(* Logix 5000 project; controller R1USB70001_CWRU_GRID_20120217 vendor 1 type 14 code 54 rev 19.11; software revision 19.01 *)

TASK MainTask (continuous, watchdog 500 ms) : MainProgram

MODULES
   Local : vendor 1 type 14 code 54 (ICP 2, rev 19.11)
      CNB_GRID : vendor 1 type 12 code 21 (ICP 0, rev 20.1)
         ACNR_GP_SC_N2 : vendor 1 type 12 code 111 (ControlNet 2, rev 1.83, Output RPI 16 ms)
            IE4C_GP_SC_S4 : 1734-IE4C (PointIO 4, rev 3.1, Input RPI 16 ms)
            IB8_GP_SC_S11 : 1734-IB8 (PointIO 11, rev 3.22)
            IE4C_GP_SC_S8 : 1734-IE4C (PointIO 8, rev 3.1, Input RPI 16 ms)
            IE4C_GP_SC_S5 : 1734-IE4C (PointIO 5, rev 3.1, Input RPI 16 ms)
            IE4C_GP_SC_S6 : 1734-IE4C (PointIO 6, rev 3.1, Input RPI 16 ms)
            IE4C_GP_SC_S9 : 1734-IE4C (PointIO 9, rev 3.1, Input RPI 16 ms)
            IE4C_GP_SC_S1 : 1734-IE4C (PointIO 1, rev 3.1, Input RPI 16 ms)
            IB8_GP_SC_S10 : 1734-IB8 (PointIO 10, rev 3.22)
            IE4C_GP_SC_S2 : 1734-IE4C (PointIO 2, rev 3.1, Input RPI 16 ms)
            IE4C_GP_SC_S7 : 1734-IE4C (PointIO 7, rev 3.1, Input RPI 16 ms)
            IE4C_GP_SC_S3 : 1734-IE4C (PointIO 3, rev 3.1, Input RPI 16 ms)
            OB8_GP_SC_S19 : 1734-OB8 (PointIO 19, rev 3.22)
            OB8_GP_SC_S13 : 1734-OB8 (PointIO 13, rev 3.22)
            OB8_GP_SC_S18 : 1734-OB8 (PointIO 18, rev 3.22)
            OB8_GP_SC_S23 : 1734-OB8 (PointIO 23, rev 3.22)
            OB8_GP_SC_S12 : 1734-OB8 (PointIO 12, rev 3.22)
            OB8_GP_SC_S20 : 1734-OB8 (PointIO 20, rev 3.22)
            OB8_GP_SC_S17 : 1734-OB8 (PointIO 17, rev 3.22)
            OB8_GP_SC_S15 : 1734-OB8 (PointIO 15, rev 3.22)
            OB8_GP_SC_S21 : 1734-OB8 (PointIO 21, rev 3.22)
            OB8_GP_SC_S22 : 1734-OB8 (PointIO 22, rev 3.22)
            OB8_GP_SC_S14 : 1734-OB8 (PointIO 14, rev 3.22)
            OB8_GP_SC_S16 : 1734-OB8 (PointIO 16, rev 3.22)
      EN2T_GRID : 1756-EN2T (ICP 1, Ethernet 10.88.0.102, rev 4.3)
END_MODULES

VAR_GLOBAL   (* controller tags *)
   AP_GP_CH_ACAM : ALIAS FOR ACNR_GP_SC_N2:1:I.Ch1Data;
   AP_GP_CH_CS : ALIAS FOR ACNR_GP_SC_N2:12:O.1;
   AP_GP_SR_ACAM : ALIAS FOR ACNR_GP_SC_N2:1:I.Ch0Data;
   AP_GP_SR_ACVT : ALIAS FOR ACNR_GP_SC_N2:9:I.Ch1Data;
   AP_GP_SR_CS : ALIAS FOR ACNR_GP_SC_N2:12:O.0;
   BT_GP_CH1_CS : ALIAS FOR ACNR_GP_SC_N2:12:O.3;
   BT_GP_CH2_CS : ALIAS FOR ACNR_GP_SC_N2:12:O.4;
   BT_GP_L1_ACAM1 : ALIAS FOR ACNR_GP_SC_N2:1:I.Ch2Data;
   BT_GP_L1_ACAM2 : ALIAS FOR ACNR_GP_SC_N2:1:I.Ch3Data;
   BT_GP_L1_DCAM : ALIAS FOR ACNR_GP_SC_N2:2:I.Ch2Data;
   BT_GP_L1_DCVS : ALIAS FOR ACNR_GP_SC_N2:10:I.2;
   BT_GP_L2_ACAM1 : ALIAS FOR ACNR_GP_SC_N2:2:I.Ch0Data;
   BT_GP_L2_DCAM : ALIAS FOR ACNR_GP_SC_N2:2:I.Ch3Data;
   BT_GP_ML_ACVT : ALIAS FOR ACNR_GP_SC_N2:9:I.Ch2Data;
   BT_GP_SR1_CS : ALIAS FOR ACNR_GP_SC_N2:12:O.6;
   BT_GP_SR2_CS : ALIAS FOR ACNR_GP_SC_N2:12:O.7;
   BT_GP_SR3_CS : ALIAS FOR ACNR_GP_SC_N2:13:O.0;
   CAP3_3_USER : BOOL;
   CAP_10_USER : BOOL;
   CAP_11_USER : BOOL;
   CAP_12_USER : BOOL;
   CAP_13_USER : BOOL;
   CAP_14_USER : BOOL;
   CAP_15_USER : BOOL;
   CAP_16_USER : BOOL;
   CAP_17_USER : BOOL;
   CAP_18_USER : BOOL;
   CAP_19_USER : BOOL;
   CAP_1_USER : BOOL;
   CAP_20_USER : BOOL;
   CAP_21_USER : BOOL;
   CAP_22_USER : BOOL;
   CAP_23_USER : BOOL;
   CAP_24_USER : BOOL;
   CAP_25_USER : BOOL;
   CAP_26_USER : BOOL;
   CAP_27_USER : BOOL;
   CAP_28_USER : BOOL;
   CAP_29_USER : BOOL;
   CAP_2_USER : BOOL;
   CAP_30_USER : BOOL;
   CAP_31_USER : BOOL;
   CAP_32_USER : BOOL;
   CAP_33_USER : BOOL;
   CAP_34_USER : BOOL;
   CAP_35_USER : BOOL;
   CAP_36_USER : BOOL;
   CAP_37_USER : BOOL;
   CAP_38_USER : BOOL;
   CAP_39_USER : BOOL;
   CAP_3_USER : BOOL;
   CAP_40_USER : BOOL;
   CAP_41_USER : BOOL;
   CAP_42_USER : BOOL;
   CAP_43_USER : BOOL;
   CAP_44_USER : BOOL;
   CAP_45_USER : BOOL;
   CAP_46_USER : BOOL;
   CAP_47_USER : BOOL;
   CAP_48_USER : BOOL;
   CAP_49_USER : BOOL;
   CAP_4_USER : BOOL;
   CAP_50_USER : BOOL;
   CAP_5_USER : BOOL;
   CAP_6_USER : BOOL;
   CAP_7_USER : BOOL;
   CAP_8_USER : BOOL;
   CAP_9_USER : BOOL;
   CAP_MAIN_USER : BOOL;
   CAP_MORE : DINT;
   CB_GP_C10_CS : ALIAS FOR ACNR_GP_SC_N2:18:O.2;
   CB_GP_C11_CS : ALIAS FOR ACNR_GP_SC_N2:18:O.3;
   CB_GP_C12_CS : ALIAS FOR ACNR_GP_SC_N2:18:O.4;
   CB_GP_C13_CS : ALIAS FOR ACNR_GP_SC_N2:18:O.5;
   CB_GP_C14_CS : ALIAS FOR ACNR_GP_SC_N2:18:O.6;
   CB_GP_C15_CS : ALIAS FOR ACNR_GP_SC_N2:18:O.7;
   CB_GP_C16_CS : ALIAS FOR ACNR_GP_SC_N2:19:O.0;
   CB_GP_C17_CS : ALIAS FOR ACNR_GP_SC_N2:19:O.1;
   CB_GP_C18_CS : ALIAS FOR ACNR_GP_SC_N2:19:O.2;
   CB_GP_C19_CS : ALIAS FOR ACNR_GP_SC_N2:19:O.3;
   CB_GP_C1_CS : ALIAS FOR ACNR_GP_SC_N2:17:O.1;
   CB_GP_C20_CS : ALIAS FOR ACNR_GP_SC_N2:19:O.4;
   CB_GP_C21_CS : ALIAS FOR ACNR_GP_SC_N2:19:O.5;
   CB_GP_C22_CS : ALIAS FOR ACNR_GP_SC_N2:19:O.6;
   CB_GP_C23_CS : ALIAS FOR ACNR_GP_SC_N2:19:O.7;
   CB_GP_C24_CS : ALIAS FOR ACNR_GP_SC_N2:20:O.0;
   CB_GP_C25_CS : ALIAS FOR ACNR_GP_SC_N2:20:O.1;
   CB_GP_C26_CS : ALIAS FOR ACNR_GP_SC_N2:20:O.2;
   CB_GP_C27_CS : ALIAS FOR ACNR_GP_SC_N2:20:O.3;
   CB_GP_C28_CS : ALIAS FOR ACNR_GP_SC_N2:20:O.4;
   CB_GP_C29_CS : ALIAS FOR ACNR_GP_SC_N2:20:O.5;
   CB_GP_C2_CS : ALIAS FOR ACNR_GP_SC_N2:17:O.2;
   CB_GP_C30_CS : ALIAS FOR ACNR_GP_SC_N2:20:O.6;
   CB_GP_C31_CS : ALIAS FOR ACNR_GP_SC_N2:20:O.7;
   CB_GP_C32_CS : ALIAS FOR ACNR_GP_SC_N2:21:O.0;
   CB_GP_C33_CS : ALIAS FOR ACNR_GP_SC_N2:21:O.1;
   CB_GP_C34_CS : ALIAS FOR ACNR_GP_SC_N2:21:O.2;
   CB_GP_C35_CS : ALIAS FOR ACNR_GP_SC_N2:21:O.3;
   CB_GP_C36_CS : ALIAS FOR ACNR_GP_SC_N2:21:O.4;
   CB_GP_C37_CS : ALIAS FOR ACNR_GP_SC_N2:21:O.5;
   CB_GP_C38_CS : ALIAS FOR ACNR_GP_SC_N2:21:O.6;
   CB_GP_C39_CS : ALIAS FOR ACNR_GP_SC_N2:21:O.7;
   CB_GP_C3_CS : ALIAS FOR ACNR_GP_SC_N2:17:O.3;
   CB_GP_C40_CS : ALIAS FOR ACNR_GP_SC_N2:22:O.0;
   CB_GP_C41_CS : ALIAS FOR ACNR_GP_SC_N2:22:O.1;
   CB_GP_C42_CS : ALIAS FOR ACNR_GP_SC_N2:22:O.2;
   CB_GP_C43_CS : ALIAS FOR ACNR_GP_SC_N2:22:O.3;
   CB_GP_C44_CS : ALIAS FOR ACNR_GP_SC_N2:22:O.4;
   CB_GP_C45_CS : ALIAS FOR ACNR_GP_SC_N2:22:O.5;
   CB_GP_C46_CS : ALIAS FOR ACNR_GP_SC_N2:22:O.6;
   CB_GP_C47_CS : ALIAS FOR ACNR_GP_SC_N2:22:O.7;
   CB_GP_C48_CS : ALIAS FOR ACNR_GP_SC_N2:23:O.0;
   CB_GP_C49_CS : ALIAS FOR ACNR_GP_SC_N2:23:O.1;
   CB_GP_C4_CS : ALIAS FOR ACNR_GP_SC_N2:17:O.4;
   CB_GP_C50_CS : ALIAS FOR ACNR_GP_SC_N2:23:O.2;
   CB_GP_C5_CS : ALIAS FOR ACNR_GP_SC_N2:17:O.5;
   CB_GP_C6_CS : ALIAS FOR ACNR_GP_SC_N2:17:O.6;
   CB_GP_C7_CS : ALIAS FOR ACNR_GP_SC_N2:17:O.7;
   CB_GP_C8_CS : ALIAS FOR ACNR_GP_SC_N2:18:O.0;
   CB_GP_C9_CS : ALIAS FOR ACNR_GP_SC_N2:18:O.1;
   CB_GP_ML_ACAM : ALIAS FOR ACNR_GP_SC_N2:9:I.Ch0Data;
   CB_GP_ML_ACVS : ALIAS FOR ACNR_GP_SC_N2:11:I.1;
   CB_GP_ML_CS : ALIAS FOR ACNR_GP_SC_N2:17:O.0;
   CL_GP_GD_ACAM : ALIAS FOR ACNR_GP_SC_N2:5:I.Ch2Data;
   CL_GP_GD_CS : ALIAS FOR ACNR_GP_SC_N2:15:O.1;
   CL_GP_SC_ACAM : ALIAS FOR ACNR_GP_SC_N2:4:I.Ch2Data;
   CL_GP_SC_CS : ALIAS FOR ACNR_GP_SC_N2:15:O.5;
   CL_GP_SF_ACAM : ALIAS FOR ACNR_GP_SC_N2:4:I.Ch3Data;
   CL_GP_SF_CS : ALIAS FOR ACNR_GP_SC_N2:15:O.4;
   CL_GP_WF_ACAM : ALIAS FOR ACNR_GP_SC_N2:5:I.Ch1Data;
   CL_GP_WF_CS : ALIAS FOR ACNR_GP_SC_N2:15:O.2;
   CL_GP_WT_ACAM : ALIAS FOR ACNR_GP_SC_N2:5:I.Ch0Data;
   CL_GP_WT_CS : ALIAS FOR ACNR_GP_SC_N2:15:O.3;
   COM_TO_GRID_CON : BOOL;
   COM_TO_SOURCE1_CON : BOOL;
   COM_TO_SOURCE2_CON : BOOL;
   COM_TO_SOURCE3_CON : BOOL;
   COM_TO_SOURCE4_CON : BOOL;
   COM_TO_WF_CON : BOOL;
   Comment : DINT[2] := ([0] := 3);
   HMI_Intfc_Read_Buffer : DINT[40] := ([0] := -1, [2] := -1, [3] := -1, [5] := -22, [7] := 1, [9] := 634, [10] := -1, [11] := -10, [12] := 13, [22] := -1, [23] := -1, [28] := 64, [29] := -1, [30] := -1, [31] := -1, [32] := -1, [33] := 39, [34] := 31, [35] := -12, [36] := 640, [37] := 9502720);
        [37].0   // AP_GP_SR_CS
        [8]   // RL_GP_SC_ACAM
        [12]   // RL_GP_WF_ACAM
        [9]   // RL_GP_SF_ACAM
        [10]   // RL_GP_WT_ACAM
        [13]   // RL_GP_GD_ACAM
        [14]   // CL_GP_SC_ACAM
        [15]   // CL_GP_SF_ACAM
        [16]   // CL_GP_WT_ACAM
        [17]   // CL_GP_WF_ACAM
        [18]   // CL_GP_GD_ACAM
        [19]   // IL_GP_SC_ACAM
        [20]   // IL_GP_SF_ACAM
        [21]   // IL_GP_WT_ACAM
        [22]   // IL_GP_WF_ACAM
        [23]   // IL_GP_GD_ACAM
        [37].1   // AP_GP_CH_CS
        [25]   // WF_GP_BT_ACAM
        [26]   // WT_GP_GD_ACAM
        [27]   // WT_GP_BT_ACAM
        [28]   // SF_GP_GD_ACAM
        [29]   // SF_GP_BT_ACAM
        [30]   // SC_GP_GD_ACAM
        [31]   // SC_GP_BT_ACAM
        [32]   // CB_GP_ML_ACAM
        [34]   // BT_GP_ML_ACVT
        [33]   // AP_GP_SR_ACVT
        [2]   // BT_GP_L1_ACAM1
        [3]   // BT_GP_L1_ACAM2
        [4]   // BT_GP_L2_ACAM1
        [6]   // BT_GP_L1_DCAM
        [7]   // BT_GP_L2_DCAM
        [37].3   // BT_GP_CH1_CS
        [0]   // AP_GP_SR_ACAM
        [1]   // AP_GP_CH_ACAM
        [24]   // WF_GP_GD_ACAM
        [36].2   // BT_GP_L1_DCVS
        [36].5   // WF_GP_ML_ACVS
        [36].6   // WT_GP_ML_ACVS
        [36].7   // SF_GP_ML_ACVS
        [36].8   // SC_GP_ML_ACVS
        [36].9   // CB_GP_ML_ACVS
        [37].4   // BT_GP_CH2_CS
        [37].6   // BT_GP_SR1_CS
        [37].7   // BT_GP_SR2_CS
        [37].8   // BT_GP_SR3_CS
        [37].11   // WF_GP_GD_CS
        [37].12   // WF_GP_BT_CS
        [37].13   // WT_GP_GD_CS
        [37].14   // WT_GP_BT_CS
        [37].16   // SF_GP_GD_CS
        [37].17   // SF_GP_BT_CS
        [37].18   // SC_GP_GD_CS
        [37].19   // SC_GP_BT_CS
        [37].20   // RL_GP_GD_CS
        [37].21   // RL_GP_WF_CS
        [37].22   // RL_GP_WT_CS
        [37].23   // RL_GP_SF_CS
        [37].24   // RL_GP_SC_CS
        [37].25   // CL_GP_GD_CS
        [37].26   // CL_GP_WF_CS
        [37].27   // CL_GP_WT_CS
        [37].28   // CL_GP_SF_CS
        [37].29   // CL_GP_SC_CS
        [37].30   // IL_GP_GD_CS
        [37].31   // IL_GP_WF_CS
        [38].0   // IL_GP_WT_CS
        [38].1   // IL_GP_SF_CS
        [38].2   // IL_GP_SC_CS
        [38].8   // CB_GP_ML_CS
        [38].9   // CB_GP_C1_CS
        [38].10   // CB_GP_C2_CS
        [38].11   // CB_GP_C3_CS
        [38].12   // CB_GP_C4_CS
        [38].13   // CB_GP_C5_CS
        [38].14   // CB_GP_C6_CS
        [38].15   // CB_GP_C7_CS
        [38].16   // CB_GP_C8_CS
        [38].17   // CB_GP_C9_CS
        [38].18   // CB_GP_C10_CS
        [38].19   // CB_GP_C11_CS
        [38].20   // CB_GP_C12_CS
        [38].21   // CB_GP_C13_CS
        [38].22   // CB_GP_C14_CS
        [38].23   // CB_GP_C15_CS
        [38].24   // CB_GP_C16_CS
        [38].25   // CB_GP_C17_CS
        [38].26   // CB_GP_C18_CS
        [38].27   // CB_GP_C19_CS
        [38].28   // CB_GP_C20_CS
        [38].29   // CB_GP_C21_CS
        [38].30   // CB_GP_C22_CS
        [38].31   // CB_GP_C23_CS
        [39].0   // CB_GP_C24_CS
        [39].1   // CB_GP_C25_CS
        [39].2   // CB_GP_C26_CS
        [39].3   // CB_GP_C27_CS
        [39].4   // CB_GP_C28_CS
        [39].5   // CB_GP_C29_CS
        [39].6   // CB_GP_C30_CS
        [39].7   // CB_GP_C31_CS
        [39].8   // CB_GP_C32_CS
        [39].9   // CB_GP_C33_CS
        [39].10   // CB_GP_C34_CS
        [39].11   // CB_GP_C35_CS
        [39].12   // CB_GP_C36_CS
        [39].13   // CB_GP_C37_CS
        [39].14   // CB_GP_C38_CS
        [39].15   // CB_GP_C39_CS
        [39].16   // CB_GP_C40_CS
        [39].17   // CB_GP_C41_CS
        [39].18   // CB_GP_C42_CS
        [39].19   // CB_GP_C43_CS
        [39].20   // CB_GP_C44_CS
        [39].21   // CB_GP_C45_CS
        [39].22   // CB_GP_C46_CS
        [39].23   // CB_GP_C47_CS
        [39].24   // CB_GP_C48_CS
        [39].25   // CB_GP_C49_CS
        [35]   // SPARE RESERVED FOR SLOT 9 CHANNEL 3
        [11]   // SPARE RESERVED FOR SLOT 3 CHANNEL 3
        [5]   // SPARE RESERVED FOR SLOT 2 CHANNEL 1
        [39].26   // CB_GP_C50_CS
   IL_GP_GD_ACAM : ALIAS FOR ACNR_GP_SC_N2:6:I.Ch3Data;
   IL_GP_GD_CS : ALIAS FOR ACNR_GP_SC_N2:15:O.6;
   IL_GP_SC_ACAM : ALIAS FOR ACNR_GP_SC_N2:5:I.Ch3Data;
   IL_GP_SC_CS : ALIAS FOR ACNR_GP_SC_N2:16:O.2;
   IL_GP_SF_ACAM : ALIAS FOR ACNR_GP_SC_N2:6:I.Ch0Data;
   IL_GP_SF_CS : ALIAS FOR ACNR_GP_SC_N2:16:O.1;
   IL_GP_WF_ACAM : ALIAS FOR ACNR_GP_SC_N2:6:I.Ch2Data;
   IL_GP_WF_CS : ALIAS FOR ACNR_GP_SC_N2:15:O.7;
   IL_GP_WT_ACAM : ALIAS FOR ACNR_GP_SC_N2:6:I.Ch1Data;
   IL_GP_WT_CS : ALIAS FOR ACNR_GP_SC_N2:16:O.0;
   IND_TO_GRID_CON : BOOL;
   IND_TO_SC_CON : BOOL;
   IND_TO_SF_CON : BOOL;
   IND_TO_SOURCE1_CON : BOOL;
   IND_TO_SOURCE2_CON : BOOL;
   IND_TO_SOURCE3_CON : BOOL;
   IND_TO_SOURCE4_CON : BOOL;
   IND_TO_WF_CON : BOOL;
   IND_TO_WT_CON : BOOL;
   OURCE1_TO_GRID_CON : BOOL;
   RES_TO_GRID_CON : BOOL;
   RES_TO_SOUCE3_CON : BOOL;
   RES_TO_SOURCE1_CON : BOOL;
   RES_TO_SOURCE2_CON : BOOL;
   RES_TO_SOURCE4_CON : BOOL;
   RES_TO_WF_CON : BOOL;
   RES_TO_WT_CON : BOOL;
   RL_GP_GD_ACAM : ALIAS FOR ACNR_GP_SC_N2:4:I.Ch1Data;
   RL_GP_GD_CS : ALIAS FOR ACNR_GP_SC_N2:14:O.4;
   RL_GP_SC_ACAM : ALIAS FOR ACNR_GP_SC_N2:3:I.Ch0Data;
   RL_GP_SC_CS : ALIAS FOR ACNR_GP_SC_N2:15:O.0;
   RL_GP_SF_ACAM : ALIAS FOR ACNR_GP_SC_N2:3:I.Ch1Data;
   RL_GP_SF_CS : ALIAS FOR ACNR_GP_SC_N2:14:O.7;
   RL_GP_WF_ACAM : ALIAS FOR ACNR_GP_SC_N2:4:I.Ch0Data;
   RL_GP_WF_CS : ALIAS FOR ACNR_GP_SC_N2:14:O.5;
   RL_GP_WT_ACAM : ALIAS FOR ACNR_GP_SC_N2:3:I.Ch2Data;
   RL_GP_WT_CS : ALIAS FOR ACNR_GP_SC_N2:14:O.6;
   SC_GP_BT_ACAM : ALIAS FOR ACNR_GP_SC_N2:8:I.Ch3Data;
   SC_GP_BT_CS : ALIAS FOR ACNR_GP_SC_N2:14:O.3;
   SC_GP_GD_ACAM : ALIAS FOR ACNR_GP_SC_N2:8:I.Ch2Data;
   SC_GP_GD_CS : ALIAS FOR ACNR_GP_SC_N2:14:O.2;
   SC_GP_ML_ACVS : ALIAS FOR ACNR_GP_SC_N2:11:I.0;
   SF_AC_VOLTAGE : DINT;
   SF_AC_VOLTAGE_RAW : DINT;
   SF_GP_BT_ACAM : ALIAS FOR ACNR_GP_SC_N2:8:I.Ch1Data;
   SF_GP_BT_CS : ALIAS FOR ACNR_GP_SC_N2:14:O.1;
   SF_GP_GD_ACAM : ALIAS FOR ACNR_GP_SC_N2:8:I.Ch0Data;
   SF_GP_GD_CS : ALIAS FOR ACNR_GP_SC_N2:14:O.0;
   SF_GP_ML_ACVS : ALIAS FOR ACNR_GP_SC_N2:10:I.7;
   SF_REG_DC_VOLTAGE : BOOL;
   SF_SP_LN_ACVT : DINT;
   SF_SP_LN_DCVS1 : BOOL;
   SF_SP_LN_DCVS2 : BOOL;
   SF_UNREG_DC_VOLTAGE : BOOL;
   SOURCE2_TO_GRID_CON : BOOL;
   SOURCE3_TO_GRID_CON : BOOL;
   SOURCE4_TO_GRID_CON : BOOL;
   WF_GP_BT_ACAM : ALIAS FOR ACNR_GP_SC_N2:7:I.Ch1Data;
   WF_GP_BT_CS : ALIAS FOR ACNR_GP_SC_N2:13:O.4;
   WF_GP_GD_ACAM : ALIAS FOR ACNR_GP_SC_N2:7:I.Ch0Data;
   WF_GP_GD_CS : ALIAS FOR ACNR_GP_SC_N2:13:O.3;
   WF_GP_ML_ACVS : ALIAS FOR ACNR_GP_SC_N2:10:I.5;
   WT_GP_BT_ACAM : ALIAS FOR ACNR_GP_SC_N2:7:I.Ch3Data;
   WT_GP_BT_CS : ALIAS FOR ACNR_GP_SC_N2:13:O.6;
   WT_GP_GD_ACAM : ALIAS FOR ACNR_GP_SC_N2:7:I.Ch2Data;
   WT_GP_GD_CS : ALIAS FOR ACNR_GP_SC_N2:13:O.5;
   WT_GP_ML_ACVS : ALIAS FOR ACNR_GP_SC_N2:10:I.6;
END_VAR

PROGRAM MainProgram   (* main routine MainRoutine *)
VAR
   BAT_AC_VOLTAGE : REAL := 0.022705764;
   BAT_AC_VOLTAGE_RAW : REAL := 31.0;
   BAT_CHARGE_AC_CURRENT : REAL;
   BAT_CHARGE_AC_CURRENT_RAW : REAL;
   BAT_CHARGE_DC_CURRENT : REAL := 6.1037e-05;
   BAT_CHARGE_DC_CURRENT_RAW : REAL := 1.0;
   BAT_SRC_AC_CURRENT1 : REAL := -0.00061037;
   BAT_SRC_AC_CURRENT1_RAW : REAL := -1.0;
   BAT_SRC_AC_CURRENT2 : REAL := -0.00061037;
   BAT_SRC_AC_CURRENT2_RAW : REAL := -1.0;
   BAT_SRC_DC_CURRENT : REAL;
   BAT_SRC_DC_CURRENT_RAW : REAL;
   BATT_SRC_CURRENT : REAL;
   CAES_CHARGE_CURRENT : REAL;
   CAES_CHARGE_CURRENT_RAW : REAL;
   CAES_SRC_CURRENT : REAL := -0.00061037;
   CAES_SRC_CURRENT_RAW : REAL := -1.0;
   CAP10_INT_REQ_CLOSE : BOOL;
   CAP10_REQ_CLOSE : BOOL;
   CAP10_REQ_OPEN : BOOL;
   CAP11_INT_REQ_CLOSE : BOOL;
   CAP11_REQ_CLOSE : BOOL;
   CAP11_REQ_OPEN : BOOL;
   CAP12_INT_REQ_CLOSE : BOOL;
   CAP12_REQ_CLOSE : BOOL;
   CAP12_REQ_OPEN : BOOL;
   CAP13_INT_REQ_CLOSE : BOOL;
   CAP13_REQ_CLOSE : BOOL;
   CAP13_REQ_OPEN : BOOL;
   CAP14_INT_REQ_CLOSE : BOOL;
   CAP14_REQ_CLOSE : BOOL;
   CAP14_REQ_OPEN : BOOL;
   CAP15_INT_REQ_CLOSE : BOOL;
   CAP15_REQ_CLOSE : BOOL;
   CAP15_REQ_OPEN : BOOL;
   CAP16_INT_REQ_CLOSE : BOOL;
   CAP16_REQ_CLOSE : BOOL;
   CAP16_REQ_OPEN : BOOL;
   CAP17_INT_REQ_CLOSE : BOOL;
   CAP17_REQ_CLOSE : BOOL;
   CAP17_REQ_OPEN : BOOL;
   CAP18_INT_REQ_CLOSE : BOOL;
   CAP18_REQ_CLOSE : BOOL;
   CAP18_REQ_OPEN : BOOL;
   CAP19_INT_REQ_CLOSE : BOOL;
   CAP19_REQ_CLOSE : BOOL;
   CAP19_REQ_OPEN : BOOL;
   CAP1_INT_REQ_CLOSE : BOOL;
   CAP1_REQ_CLOSE : BOOL;
   CAP1_REQ_OPEN : BOOL;
   CAP20_INT_REQ_CLOSE : BOOL;
   CAP20_REQ_CLOSE : BOOL;
   CAP20_REQ_OPEN : BOOL;
   CAP21_INT_REQ_CLOSE : BOOL;
   CAP21_REQ_CLOSE : BOOL;
   CAP21_REQ_OPEN : BOOL;
   CAP22_INT_REQ_CLOSE : BOOL;
   CAP22_REQ_CLOSE : BOOL;
   CAP22_REQ_OPEN : BOOL;
   CAP23_INT_REQ_CLOSE : BOOL;
   CAP23_REQ_CLOSE : BOOL;
   CAP23_REQ_OPEN : BOOL;
   CAP24_INT_REQ_CLOSE : BOOL;
   CAP24_REQ_CLOSE : BOOL;
   CAP24_REQ_OPEN : BOOL;
   CAP25_INT_REQ_CLOSE : BOOL;
   CAP25_REQ_CLOSE : BOOL;
   CAP25_REQ_OPEN : BOOL;
   CAP26_INT_REQ_CLOSE : BOOL;
   CAP26_REQ_CLOSE : BOOL;
   CAP26_REQ_OPEN : BOOL;
   CAP27_INT_REQ_CLOSE : BOOL;
   CAP27_REQ_CLOSE : BOOL;
   CAP27_REQ_OPEN : BOOL;
   CAP28_INT_REQ_CLOSE : BOOL;
   CAP28_REQ_CLOSE : BOOL;
   CAP28_REQ_OPEN : BOOL;
   CAP29_INT_REQ_CLOSE : BOOL;
   CAP29_REQ_CLOSE : BOOL;
   CAP29_REQ_OPEN : BOOL;
   CAP2_INT_REQ_CLOSE : BOOL;
   CAP2_REQ_CLOSE : BOOL;
   CAP2_REQ_OPEN : BOOL;
   CAP30_INT_REQ_CLOSE : BOOL;
   CAP30_REQ_CLOSE : BOOL;
   CAP30_REQ_OPEN : BOOL;
   CAP31_INT_REQ_CLOSE : BOOL;
   CAP31_REQ_CLOSE : BOOL;
   CAP31_REQ_OPEN : BOOL;
   CAP32_INT_REQ_CLOSE : BOOL;
   CAP32_REQ_CLOSE : BOOL;
   CAP32_REQ_OPEN : BOOL;
   CAP33_INT_REQ_CLOSE : BOOL;
   CAP33_REQ_CLOSE : BOOL;
   CAP33_REQ_OPEN : BOOL;
   CAP34_INT_REQ_CLOSE : BOOL;
   CAP34_REQ_CLOSE : BOOL;
   CAP34_REQ_OPEN : BOOL;
   CAP35_INT_REQ_CLOSE : BOOL;
   CAP35_REQ_CLOSE : BOOL;
   CAP35_REQ_OPEN : BOOL;
   CAP36_INT_REQ_CLOSE : BOOL;
   CAP36_REQ_CLOSE : BOOL;
   CAP36_REQ_OPEN : BOOL;
   CAP37_INT_REQ_CLOSE : BOOL;
   CAP37_REQ_CLOSE : BOOL;
   CAP37_REQ_OPEN : BOOL;
   CAP38_INT_REQ_CLOSE : BOOL;
   CAP38_REQ_CLOSE : BOOL;
   CAP38_REQ_OPEN : BOOL;
   CAP39_INT_REQ_CLOSE : BOOL;
   CAP39_REQ_CLOSE : BOOL;
   CAP39_REQ_OPEN : BOOL;
   CAP3_INT_REQ_CLOSE : BOOL;
   CAP3_REQ_CLOSE : BOOL;
   CAP3_REQ_OPEN : BOOL;
   CAP40_INT_REQ_CLOSE : BOOL;
   CAP40_REQ_CLOSE : BOOL;
   CAP40_REQ_OPEN : BOOL;
   CAP41_INT_REQ_CLOSE : BOOL;
   CAP41_REQ_CLOSE : BOOL;
   CAP41_REQ_OPEN : BOOL;
   CAP42_INT_REQ_CLOSE : BOOL;
   CAP42_REQ_CLOSE : BOOL;
   CAP42_REQ_OPEN : BOOL;
   CAP43_INT_REQ_CLOSE : BOOL;
   CAP43_REQ_CLOSE : BOOL;
   CAP43_REQ_OPEN : BOOL;
   CAP44_INT_REQ_CLOSE : BOOL;
   CAP44_REQ_CLOSE : BOOL;
   CAP44_REQ_OPEN : BOOL;
   CAP45_INT_REQ_CLOSE : BOOL;
   CAP45_REQ_CLOSE : BOOL;
   CAP45_REQ_OPEN : BOOL;
   CAP46_INT_REQ_CLOSE : BOOL;
   CAP46_REQ_CLOSE : BOOL;
   CAP46_REQ_OPEN : BOOL;
   CAP47_INT_REQ_CLOSE : BOOL;
   CAP47_REQ_CLOSE : BOOL;
   CAP47_REQ_OPEN : BOOL;
   CAP48_INT_REQ_CLOSE : BOOL;
   CAP48_REQ_CLOSE : BOOL;
   CAP48_REQ_OPEN : BOOL;
   CAP49_INT_REQ_CLOSE : BOOL;
   CAP49_REQ_CLOSE : BOOL;
   CAP49_REQ_OPEN : BOOL;
   CAP4_INT_REQ_CLOSE : BOOL;
   CAP4_REQ_CLOSE : BOOL;
   CAP4_REQ_OPEN : BOOL;
   CAP50_INT_REQ_CLOSE : BOOL;
   CAP50_REQ_CLOSE : BOOL;
   CAP50_REQ_OPEN : BOOL;
   CAP5_INT_REQ_CLOSE : BOOL;
   CAP5_REQ_CLOSE : BOOL;
   CAP5_REQ_OPEN : BOOL;
   CAP6_INT_REQ_CLOSE : BOOL;
   CAP6_REQ_CLOSE : BOOL;
   CAP6_REQ_OPEN : BOOL;
   CAP7_INT_REQ_CLOSE : BOOL;
   CAP7_REQ_CLOSE : BOOL;
   CAP7_REQ_OPEN : BOOL;
   CAP8_INT_REQ_CLOSE : BOOL;
   CAP8_REQ_CLOSE : BOOL;
   CAP8_REQ_OPEN : BOOL;
   CAP9_INT_REQ_CLOSE : BOOL;
   CAP9_REQ_CLOSE : BOOL;
   CAP9_REQ_OPEN : BOOL;
   CAP_MAIN_CURRENT : REAL := -0.00061037;
   CAP_MAIN_CURRENT_RAW : REAL := -1.0;
   CAP_MAIN_INT_REQ_CLOSE : BOOL;
   CAP_MAIN_REQ_CLOSE : BOOL;
   CAP_MAIN_REQ_OPEN : BOOL;
   COM_HighVoltage : BOOL;
   COM_HighVoltageThreshold : REAL;
   COM_LowVoltage : BOOL;
   COM_LowVoltageThreshold : REAL;
   COM_TO_GRID_CLOSE_FAIL : BOOL;
   COM_TO_GRID_CLOSE_FAIL_THRESH : REAL;
   COM_TO_GRID_CLOSE_PROXY : BOOL;
   COM_TO_GRID_CLOSED : BOOL;
   COM_TO_GRID_COMMAND_CHANGED : BOOL;
   COM_TO_GRID_COMMAND_CHANGED_TIMER : TIMER := (PRE := 5000);
   COM_TO_GRID_CURRENT : REAL;
   COM_TO_GRID_CURRENT_RAW : REAL;
   COM_TO_GRID_INT_REQ_CLOSE : BOOL;
   COM_TO_GRID_INT_REQ_CONNECT : BOOL;
   COM_TO_GRID_OPEN_FAIL : BOOL := 1;
   COM_TO_GRID_OPEN_FAIL_THRESH : REAL;
   COM_TO_GRID_REQ_CLOSE : BOOL;
   COM_TO_GRID_REQ_CONNECT : BOOL;
   COM_TO_GRID_REQ_DISCONNECT : BOOL;
   COM_TO_GRID_REQ_OPEN : BOOL := 1;
   COM_TO_SC_CLOSE_FAIL : BOOL;
   COM_TO_SC_CLOSE_FAIL_THRESH : REAL;
   COM_TO_SC_CLOSE_PROXY : BOOL;
   COM_TO_SC_CLOSED : BOOL;
   COM_TO_SC_COMMAND_CHANGED : BOOL;
   COM_TO_SC_COMMAND_CHANGED_TIMER : TIMER := (PRE := 5000);
   COM_TO_SC_INT_REQ_CLOSE : BOOL;
   COM_TO_SC_INT_REQ_CONNECT : BOOL;
   COM_TO_SC_OPEN_FAIL : BOOL := 1;
   COM_TO_SC_OPEN_FAIL_THRESH : REAL;
   COM_TO_SC_REQ_CLOSE : BOOL;
   COM_TO_SC_REQ_CONNECT : BOOL;
   COM_TO_SC_REQ_DISCONNECT : BOOL;
   COM_TO_SC_REQ_OPEN : BOOL := 1;
   COM_TO_SF_CLOSE_FAIL : BOOL;
   COM_TO_SF_CLOSE_FAIL_THRESH : REAL;
   COM_TO_SF_CLOSE_PROXY : BOOL;
   COM_TO_SF_CLOSED : BOOL;
   COM_TO_SF_COMMAND_CHANGED : BOOL;
   COM_TO_SF_COMMAND_CHANGED_TIMER : TIMER := (PRE := 5000);
   COM_TO_SF_INT_REQ_CLOSE : BOOL;
   COM_TO_SF_INT_REQ_CONNECT : BOOL;
   COM_TO_SF_OPEN_FAIL : BOOL := 1;
   COM_TO_SF_OPEN_FAIL_THRESH : REAL;
   COM_TO_SF_REQ_CLOSE : BOOL;
   COM_TO_SF_REQ_CONNECT : BOOL;
   COM_TO_SF_REQ_DISCONNECT : BOOL;
   COM_TO_SF_REQ_OPEN : BOOL := 1;
   COM_TO_WF_CLOSE_FAIL : BOOL;
   COM_TO_WF_CLOSE_FAIL_THRESH : REAL;
   COM_TO_WF_CLOSE_PROXY : BOOL;
   COM_TO_WF_CLOSED : BOOL;
   COM_TO_WF_COMMAND_CHANGED : BOOL;
   COM_TO_WF_COMMAND_CHANGED_TIMER : TIMER := (PRE := 5000);
   COM_TO_WF_INT_REQ_CLOSE : BOOL;
   COM_TO_WF_INT_REQ_CONNECT : BOOL;
   COM_TO_WF_OPEN_FAIL : BOOL := 1;
   COM_TO_WF_OPEN_FAIL_THRESH : REAL;
   COM_TO_WF_REQ_CLOSE : BOOL;
   COM_TO_WF_REQ_CONNECT : BOOL;
   COM_TO_WF_REQ_DISCONNECT : BOOL;
   COM_TO_WF_REQ_OPEN : BOOL := 1;
   COM_TO_WT_CLOSE_FAIL : BOOL;
   COM_TO_WT_CLOSE_FAIL_THRESH : REAL;
   COM_TO_WT_CLOSE_PROXY : BOOL;
   COM_TO_WT_CLOSED : BOOL;
   COM_TO_WT_COMMAND_CHANGED : BOOL;
   COM_TO_WT_COMMAND_CHANGED_TIMER : TIMER;
   COM_TO_WT_INT_REQ_CLOSE : BOOL;
   COM_TO_WT_INT_REQ_CONNECT : BOOL;
   COM_TO_WT_OPEN_FAIL : BOOL := 1;
   COM_TO_WT_OPEN_FAIL_THRESH : REAL;
   COM_TO_WT_REQ_CLOSE : BOOL;
   COM_TO_WT_REQ_CONNECT : BOOL;
   COM_TO_WT_REQ_DISCONNECT : BOOL;
   COM_TO_WT_REQ_OPEN : BOOL := 1;
   CURRENT_SCALE_HIGH : REAL := 0.00061037;
   CURRENT_SCALE_LOW : REAL := 6.1037e-05;
   FEWER_CAPACITORS : BOOL;
   IND_HighVoltage : BOOL;
   IND_LowVoltage : BOOL;
   IND_LowVoltageThreshold : REAL;
   IND_TO_GRID_CLOSE_FAIL : BOOL;
   IND_TO_GRID_CLOSE_FAIL_THRESH : REAL;
   IND_TO_GRID_CLOSE_PROXY : BOOL;
   IND_TO_GRID_CLOSED : BOOL;
   IND_TO_GRID_COMMAND_CHANGED : BOOL;
   IND_TO_GRID_COMMAND_CHANGED_TIMER : TIMER := (PRE := 5000);
   IND_TO_GRID_CURRENT : REAL := -0.00061037;
   IND_TO_GRID_CURRENT_RAW : REAL := -1.0;
   IND_TO_GRID_INT_REQ_CLOSE : BOOL;
   IND_TO_GRID_INT_REQ_CONNECT : BOOL;
   IND_TO_GRID_OPEN_FAIL : BOOL;
   IND_TO_GRID_OPEN_FAIL_THRESH : REAL;
   IND_TO_GRID_REQ_CLOSE : BOOL;
   IND_TO_GRID_REQ_CONNECT : BOOL;
   IND_TO_GRID_REQ_DISCONNECT : BOOL;
   IND_TO_GRID_REQ_OPEN : BOOL := 1;
   IND_TO_SC_CLOSE_FAIL : BOOL;
   IND_TO_SC_CLOSE_PROXY : BOOL;
   IND_TO_SC_CLOSED : BOOL;
   IND_TO_SC_COMMAND_CHANGED : BOOL;
   IND_TO_SC_COMMAND_CHANGED_TIMER : TIMER := (PRE := 5000);
   IND_TO_SC_INT_REQ_CLOSE : BOOL;
   IND_TO_SC_INT_REQ_CONNECT : BOOL;
   IND_TO_SC_OPEN_FAIL : BOOL;
   IND_TO_SC_REQ_CLOSE : BOOL;
   IND_TO_SC_REQ_CONNECT : BOOL;
   IND_TO_SC_REQ_DISCONNECT : BOOL;
   IND_TO_SC_REQ_OPEN : BOOL := 1;
   IND_TO_SF_CLOSE_FAIL : BOOL;
   IND_TO_SF_CLOSE_FAIL_THRESH : REAL;
   IND_TO_SF_CLOSE_PROXY : BOOL;
   IND_TO_SF_CLOSED : BOOL;
   IND_TO_SF_COMMAND_CHANGED : BOOL;
   IND_TO_SF_COMMAND_CHANGED_TIMER : TIMER := (PRE := 5000);
   IND_TO_SF_INT_REQ_CLOSE : BOOL;
   IND_TO_SF_INT_REQ_CONNECT : BOOL;
   IND_TO_SF_OPEN_FAIL : BOOL := 1;
   IND_TO_SF_OPEN_FAIL_THRESH : REAL;
   IND_TO_SF_REQ_CLOSE : BOOL;
   IND_TO_SF_REQ_CONNECT : BOOL;
   IND_TO_SF_REQ_DISCONNECT : BOOL;
   IND_TO_SF_REQ_OPEN : BOOL := 1;
   IND_TO_WF_CLOSE_FAIL : BOOL;
   IND_TO_WF_CLOSE_FAIL_THRESH : REAL;
   IND_TO_WF_CLOSE_PROXY : BOOL;
   IND_TO_WF_CLOSED : BOOL;
   IND_TO_WF_COMMAND_CHANGED : BOOL;
   IND_TO_WF_COMMAND_CHANGED_TIMER : TIMER := (PRE := 5000);
   IND_TO_WF_INT_REQ_CLOSE : BOOL;
   IND_TO_WF_INT_REQ_CONNECT : BOOL;
   IND_TO_WF_OPEN_FAIL : BOOL;
   IND_TO_WF_OPEN_FAIL_THRESH : REAL;
   IND_TO_WF_REQ_CLOSE : BOOL;
   IND_TO_WF_REQ_CONNECT : BOOL;
   IND_TO_WF_REQ_DISCONNECT : BOOL;
   IND_TO_WF_REQ_OPEN : BOOL := 1;
   IND_TO_WT_CLOSE_FAIL : BOOL;
   IND_TO_WT_CLOSE_FAIL_THRESH : REAL;
   IND_TO_WT_CLOSE_PROXY : BOOL;
   IND_TO_WT_CLOSED : BOOL;
   IND_TO_WT_COMMAND_CHANGED : BOOL;
   IND_TO_WT_COMMAND_CHANGED_TIMER : TIMER;
   IND_TO_WT_INT_REQ_CLOSE : BOOL;
   IND_TO_WT_INT_REQ_CONNECT : BOOL;
   IND_TO_WT_OPEN_FAIL : BOOL := 1;
   IND_TO_WT_OPEN_FAIL_THRESH : REAL;
   IND_TO_WT_REQ_CLOSE : BOOL;
   IND_TO_WT_REQ_CONNECT : BOOL;
   IND_TO_WT_REQ_DISCONNECT : BOOL;
   IND_TO_WT_REQ_OPEN : BOOL := 1;
   INITIALIZE_GRID : BOOL;
   INITIALIZE_GUARD : BOOL;
   INITIALIZE_GUARD_INT : BOOL;
   MAINS_AC_VOLTAGE : REAL := 0.028565316;
   MAINS_AC_VOLTAGE_RAW : REAL := 39.0;
   MORE_CAPACITORS : BOOL;
   OkToConnect : BOOL;
   PF_LOWER_LIM : REAL;
   PF_UPPER_LIM : REAL;
   POWER_FACTOR : REAL;
   RES_HighVoltage : BOOL;
   RES_HighVoltageThreshold : REAL;
   RES_LowVoltage : BOOL;
   RES_LowVoltageThreshold : REAL;
   RES_TO_GRID_CLOSE_FAIL : BOOL := 1;
   RES_TO_GRID_CLOSE_FAIL_THRESH : REAL;
   RES_TO_GRID_CLOSE_PROXY : BOOL := 1;
   RES_TO_GRID_CLOSED : BOOL := 1;
   RES_TO_GRID_COMMAND_CHANGED : BOOL;
   RES_TO_GRID_COMMAND_CHANGED_TIMER : TIMER := (PRE := 5000);
   RES_TO_GRID_CURRENT : REAL;
   RES_TO_GRID_CURRENT_RAW : REAL;
   RES_TO_GRID_INT_REQ_CLOSE : BOOL := 1;
   RES_TO_GRID_INT_REQ_CONNECT : BOOL := 1;
   RES_TO_GRID_OPEN_FAIL : BOOL;
   RES_TO_GRID_OPEN_FAIL_THRESH : REAL;
   RES_TO_GRID_REQ_CLOSE : BOOL := 1;
   RES_TO_GRID_REQ_CONNECT : BOOL := 1;
   RES_TO_GRID_REQ_DISCONNECT : BOOL;
   RES_TO_GRID_REQ_OPEN : BOOL;
   RES_TO_SC_CLOSE_FAIL : BOOL;
   RES_TO_SC_CLOSE_FAIL_THRESH : REAL;
   RES_TO_SC_CLOSE_PROXY : BOOL;
   RES_TO_SC_CLOSED : BOOL;
   RES_TO_SC_COMMAND_CHANGED : BOOL;
   RES_TO_SC_COMMAND_CHANGED_TIMER : TIMER := (PRE := 5000);
   RES_TO_SC_INT_REQ_CLOSE : BOOL;
   RES_TO_SC_INT_REQ_CONNECT : BOOL;
   RES_TO_SC_OPEN_FAIL : BOOL := 1;
   RES_TO_SC_OPEN_FAIL_THRESH : REAL;
   RES_TO_SC_REQ_CLOSE : BOOL;
   RES_TO_SC_REQ_CONNECT : BOOL;
   RES_TO_SC_REQ_DISCONNECT : BOOL;
   RES_TO_SC_REQ_OPEN : BOOL := 1;
   RES_TO_SF_CLOSE_FAIL : BOOL;
   RES_TO_SF_CLOSE_FAIL_THRESH : REAL;
   RES_TO_SF_CLOSE_PROXY : BOOL := 1;
   RES_TO_SF_CLOSED : BOOL := 1;
   RES_TO_SF_COMMAND_CHANGED : BOOL := 1;
   RES_TO_SF_COMMAND_CHANGED_TIMER : TIMER := (PRE := 5000, ACC := 1, EN := 1, TT := 1);
   RES_TO_SF_INT_REQ_CLOSE : BOOL := 1;
   RES_TO_SF_INT_REQ_CONNECT : BOOL := 1;
   RES_TO_SF_OPEN_FAIL : BOOL;
   RES_TO_SF_OPEN_FAIL_THRESH : REAL;
   RES_TO_SF_REQ_CLOSE : BOOL := 1;
   RES_TO_SF_REQ_CONNECT : BOOL;
   RES_TO_SF_REQ_DISCONNECT : BOOL;
   RES_TO_SF_REQ_OPEN : BOOL;
   RES_TO_WF_CLOSE_FAIL : BOOL;
   RES_TO_WF_CLOSE_FAIL_THRESH : REAL;
   RES_TO_WF_CLOSE_PROXY : BOOL;
   RES_TO_WF_CLOSED : BOOL;
   RES_TO_WF_COMMAND_CHANGED : BOOL;
   RES_TO_WF_COMMAND_CHANGED_TIMER : TIMER := (PRE := 5000);
   RES_TO_WF_INT_REQ_CLOSE : BOOL;
   RES_TO_WF_INT_REQ_CONNECT : BOOL;
   RES_TO_WF_OPEN_FAIL : BOOL := 1;
   RES_TO_WF_OPEN_FAIL_THRESH : REAL;
   RES_TO_WF_REQ_CLOSE : BOOL;
   RES_TO_WF_REQ_CONNECT : BOOL;
   RES_TO_WF_REQ_DISCONNECT : BOOL;
   RES_TO_WF_REQ_OPEN : BOOL := 1;
   RES_TO_WT_CLOSE_FAIL : BOOL;
   RES_TO_WT_CLOSE_FAIL_THRESH : REAL;
   RES_TO_WT_CLOSE_PROXY : BOOL;
   RES_TO_WT_CLOSED : BOOL;
   RES_TO_WT_COMMAND_CHANGED : BOOL;
   RES_TO_WT_COMMAND_CHANGED_TIMER : TIMER := (PRE := 5000);
   RES_TO_WT_INT_REQ_CLOSE : BOOL;
   RES_TO_WT_INT_REQ_CONNECT : BOOL;
   RES_TO_WT_OPEN_FAIL : BOOL;
   RES_TO_WT_OPEN_FAIL_THRESH : REAL;
   RES_TO_WT_REQ_CLOSE : BOOL;
   RES_TO_WT_REQ_CONNECT : BOOL;
   RES_TO_WT_REQ_DISCONNECT : BOOL;
   RES_TO_WT_REQ_OPEN : BOOL := 1;
   SC_TO_BAT_CURRENT : REAL := -0.00061037;
   SC_TO_BAT_CURRENT_RAW : REAL := -1.0;
   SC_TO_COM_CURRENT : REAL;
   SC_TO_COM_CURRENT_RAW : REAL;
   SC_TO_GRID_CLOSE_FAIL : BOOL;
   SC_TO_GRID_CLOSE_FAIL_THRESH : REAL;
   SC_TO_GRID_CLOSE_PROXY : BOOL;
   SC_TO_GRID_CLOSED : BOOL;
   SC_TO_GRID_COMMAND_CHANGED : BOOL;
   SC_TO_GRID_COMMAND_CHANGED_TIMER : TIMER := (PRE := 5000);
   SC_TO_GRID_CURRENT : REAL := -0.00061037;
   SC_TO_GRID_CURRENT_RAW : REAL := -1.0;
   SC_TO_GRID_INT_REQ_CLOSE : BOOL;
   SC_TO_GRID_INT_REQ_CONNECT : BOOL;
   SC_TO_GRID_OPEN_FAIL : BOOL;
   SC_TO_GRID_OPEN_FAIL_THRESH : REAL;
   SC_TO_GRID_REQ_CLOSE : BOOL;
   SC_TO_GRID_REQ_CONNECT : BOOL;
   SC_TO_GRID_REQ_DISCONNECT : BOOL;
   SC_TO_GRID_REQ_OPEN : BOOL := 1;
   SC_TO_IND_CLOSE_FAIL_THRESH : REAL;
   SC_TO_IND_CURRENT : REAL;
   SC_TO_IND_CURRENT_RAW : REAL;
   SC_TO_IND_OPEN_FAIL_THRESH : REAL := 0.02;
   SC_TO_RES_CURRENT : REAL;
   SC_TO_RES_CURRENT_RAW : REAL;
   SF_POWER_AVAILABLE : BOOL;
   SF_TO_BAT_CURRENT : REAL := -0.00061037;
   SF_TO_BAT_CURRENT_RAW : REAL := -1.0;
   SF_TO_COM_CURRENT : REAL;
   SF_TO_COM_CURRENT_RAW : REAL;
   SF_TO_GRID_CLOSE_FAIL : BOOL;
   SF_TO_GRID_CLOSE_FAIL_THRESH : REAL := 0.02;
   SF_TO_GRID_CLOSE_PROXY : BOOL := 1;
   SF_TO_GRID_CLOSED : BOOL := 1;
   SF_TO_GRID_COMMAND_CHANGED : BOOL;
   SF_TO_GRID_COMMAND_CHANGED_TIMER : TIMER := (PRE := 2000);
   SF_TO_GRID_CURRENT : REAL := 0.03906368;
   SF_TO_GRID_CURRENT_RAW : REAL := 64.0;
   SF_TO_GRID_INT_REQ_CLOSE : BOOL := 1;
   SF_TO_GRID_INT_REQ_CONNECT : BOOL := 1;
   SF_TO_GRID_OPEN_FAIL : BOOL;
   SF_TO_GRID_OPEN_FAIL_THRESH : REAL;
   SF_TO_GRID_REQ_CLOSE : BOOL := 1;
   SF_TO_GRID_REQ_CONNECT : BOOL := 1;
   SF_TO_GRID_REQ_DISCONNECT : BOOL;
   SF_TO_GRID_REQ_OPEN : BOOL;
   SF_TO_IND_CURRENT : REAL;
   SF_TO_IND_CURRENT_RAW : REAL;
   SF_TO_RES_CURRENT : REAL := 0.3869746;
   SF_TO_RES_CURRENT_RAW : REAL := 634.0;
   TOTAL_CAP_DEMAND : DINT;
   VOLTAGE_SCALE : REAL := 0.000732444;
   WF_TO_BAT_CURRENT : REAL;
   WF_TO_BAT_CURRENT_RAW : REAL;
   WF_TO_COM_CURRENT : REAL;
   WF_TO_COM_CURRENT_RAW : REAL;
   WF_TO_GRID_CLOSE_FAIL : BOOL;
   WF_TO_GRID_CLOSE_FAIL_THRESH : REAL;
   WF_TO_GRID_CLOSE_PROXY : BOOL;
   WF_TO_GRID_CLOSED : BOOL;
   WF_TO_GRID_COMMAND_CHANGED : BOOL;
   WF_TO_GRID_COMMAND_CHANGED_TIMER : TIMER := (PRE := 5000);
   WF_TO_GRID_CURRENT : REAL;
   WF_TO_GRID_CURRENT_RAW : REAL;
   WF_TO_GRID_INT_REQ_CLOSE : BOOL;
   WF_TO_GRID_INT_REQ_CONNECT : BOOL;
   WF_TO_GRID_OPEN_FAIL : BOOL := 1;
   WF_TO_GRID_OPEN_FAIL_THRESH : REAL;
   WF_TO_GRID_REQ_CLOSE : BOOL;
   WF_TO_GRID_REQ_CONNECT : BOOL;
   WF_TO_GRID_REQ_DISCONNECT : BOOL;
   WF_TO_GRID_REQ_OPEN : BOOL := 1;
   WF_TO_IND_CURRENT : REAL := -0.00061037;
   WF_TO_IND_CURRENT_RAW : REAL := -1.0;
   WF_TO_RES_CURRENT : REAL := 0.007934811;
   WF_TO_RES_CURRENT_RAW : REAL := 13.0;
   WT_TO_BAT_CURRENT : REAL;
   WT_TO_BAT_CURRENT_RAW : REAL;
   WT_TO_COM_CURRENT : REAL;
   WT_TO_COM_CURRENT_RAW : REAL;
   WT_TO_GRID_CLOSE_FAIL : BOOL;
   WT_TO_GRID_CLOSE_FAIL_THRESH : REAL;
   WT_TO_GRID_CLOSE_PROXY : BOOL;
   WT_TO_GRID_CLOSED : BOOL;
   WT_TO_GRID_COMMAND_CHANGED : BOOL;
   WT_TO_GRID_COMMAND_CHANGED_TIMER : TIMER := (PRE := 5000);
   WT_TO_GRID_CURRENT : REAL;
   WT_TO_GRID_CURRENT_RAW : REAL;
   WT_TO_GRID_INT_REQ_CLOSE : BOOL;
   WT_TO_GRID_INT_REQ_CONNECT : BOOL;
   WT_TO_GRID_OPEN_FAIL : BOOL := 1;
   WT_TO_GRID_OPEN_FAIL_THRESH : REAL;
   WT_TO_GRID_REQ_CLOSE : BOOL;
   WT_TO_GRID_REQ_CONNECT : BOOL;
   WT_TO_GRID_REQ_DISCONNECT : BOOL;
   WT_TO_GRID_REQ_OPEN : BOOL := 1;
   WT_TO_IND_CURRENT : REAL;
   WT_TO_IND_CURRENT_RAW : REAL;
   WT_TO_RES_CURRENT : REAL := -0.00061037;
   WT_TO_RES_CURRENT_RAW : REAL := -1.0;
END_VAR

ROUTINE CapBankManagement   (* ladder *)
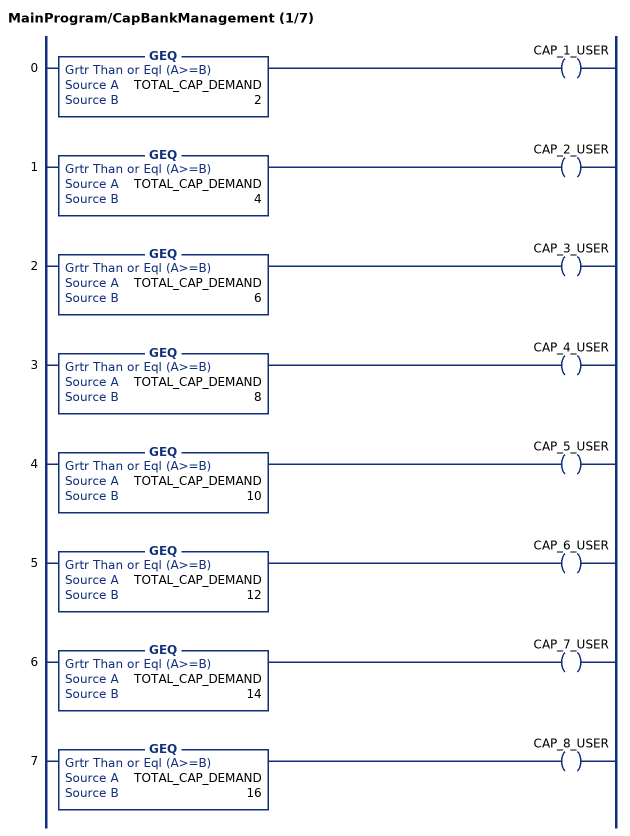
   0: GEQ(TOTAL_CAP_DEMAND,2)OTE(CAP_1_USER);
   1: GEQ(TOTAL_CAP_DEMAND,4)OTE(CAP_2_USER);
   2: GEQ(TOTAL_CAP_DEMAND,6)OTE(CAP_3_USER);
   3: GEQ(TOTAL_CAP_DEMAND,8)OTE(CAP_4_USER);
   4: GEQ(TOTAL_CAP_DEMAND,10)OTE(CAP_5_USER);
   5: GEQ(TOTAL_CAP_DEMAND,12)OTE(CAP_6_USER);
   6: GEQ(TOTAL_CAP_DEMAND,14)OTE(CAP_7_USER);
   7: GEQ(TOTAL_CAP_DEMAND,16)OTE(CAP_8_USER);
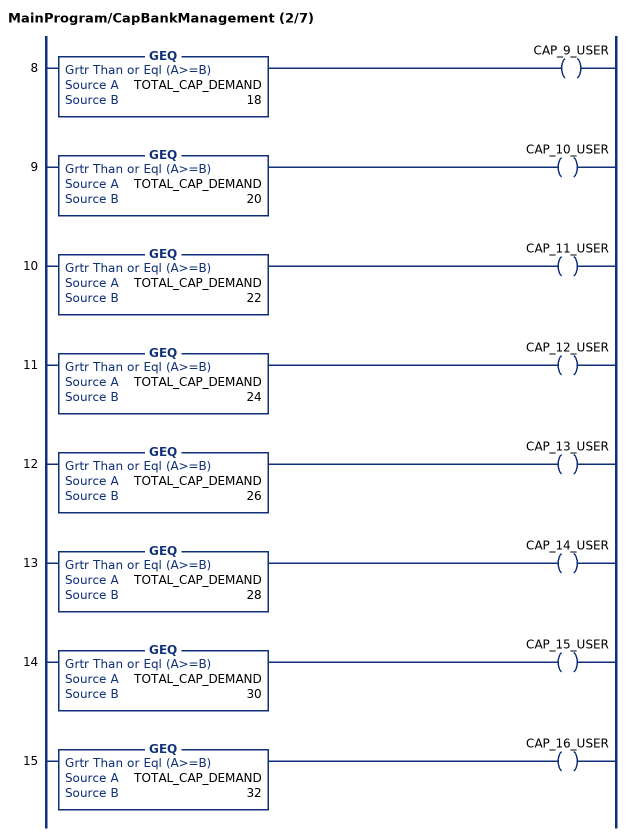
   8: GEQ(TOTAL_CAP_DEMAND,18)OTE(CAP_9_USER);
   9: GEQ(TOTAL_CAP_DEMAND,20)OTE(CAP_10_USER);
   10: GEQ(TOTAL_CAP_DEMAND,22)OTE(CAP_11_USER);
   11: GEQ(TOTAL_CAP_DEMAND,24)OTE(CAP_12_USER);
   12: GEQ(TOTAL_CAP_DEMAND,26)OTE(CAP_13_USER);
   13: GEQ(TOTAL_CAP_DEMAND,28)OTE(CAP_14_USER);
   14: GEQ(TOTAL_CAP_DEMAND,30)OTE(CAP_15_USER);
   15: GEQ(TOTAL_CAP_DEMAND,32)OTE(CAP_16_USER);
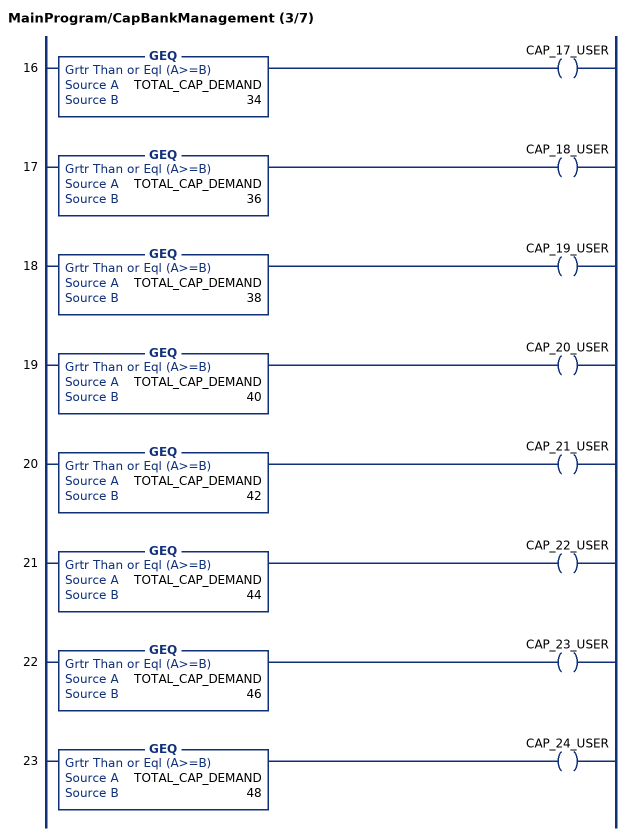
   16: GEQ(TOTAL_CAP_DEMAND,34)OTE(CAP_17_USER);
   17: GEQ(TOTAL_CAP_DEMAND,36)OTE(CAP_18_USER);
   18: GEQ(TOTAL_CAP_DEMAND,38)OTE(CAP_19_USER);
   19: GEQ(TOTAL_CAP_DEMAND,40)OTE(CAP_20_USER);
   20: GEQ(TOTAL_CAP_DEMAND,42)OTE(CAP_21_USER);
   21: GEQ(TOTAL_CAP_DEMAND,44)OTE(CAP_22_USER);
   22: GEQ(TOTAL_CAP_DEMAND,46)OTE(CAP_23_USER);
   23: GEQ(TOTAL_CAP_DEMAND,48)OTE(CAP_24_USER);
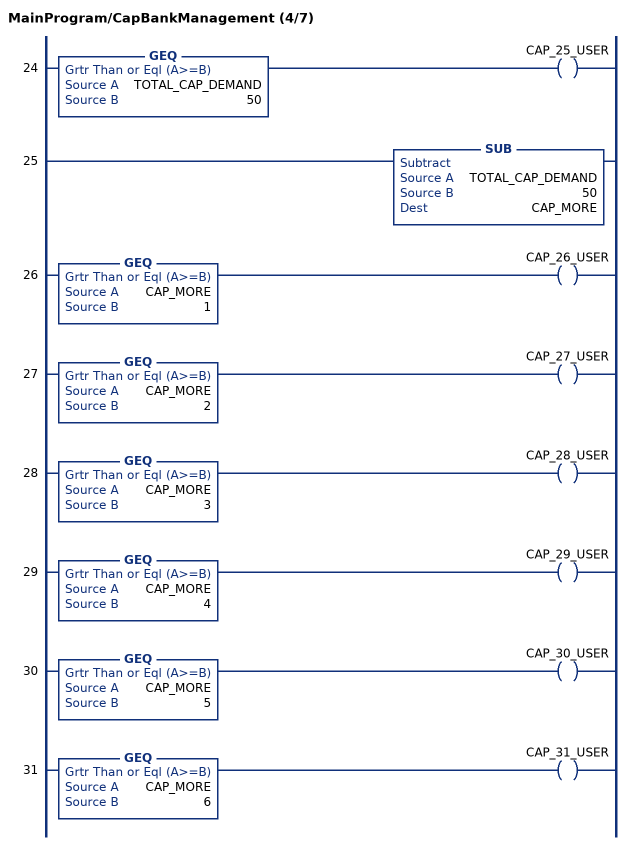
   24: GEQ(TOTAL_CAP_DEMAND,50)OTE(CAP_25_USER);
   25: SUB(TOTAL_CAP_DEMAND,50,CAP_MORE);
   26: GEQ(CAP_MORE,1)OTE(CAP_26_USER);
   27: GEQ(CAP_MORE,2)OTE(CAP_27_USER);
   28: GEQ(CAP_MORE,3)OTE(CAP_28_USER);
   29: GEQ(CAP_MORE,4)OTE(CAP_29_USER);
   30: GEQ(CAP_MORE,5)OTE(CAP_30_USER);
   31: GEQ(CAP_MORE,6)OTE(CAP_31_USER);
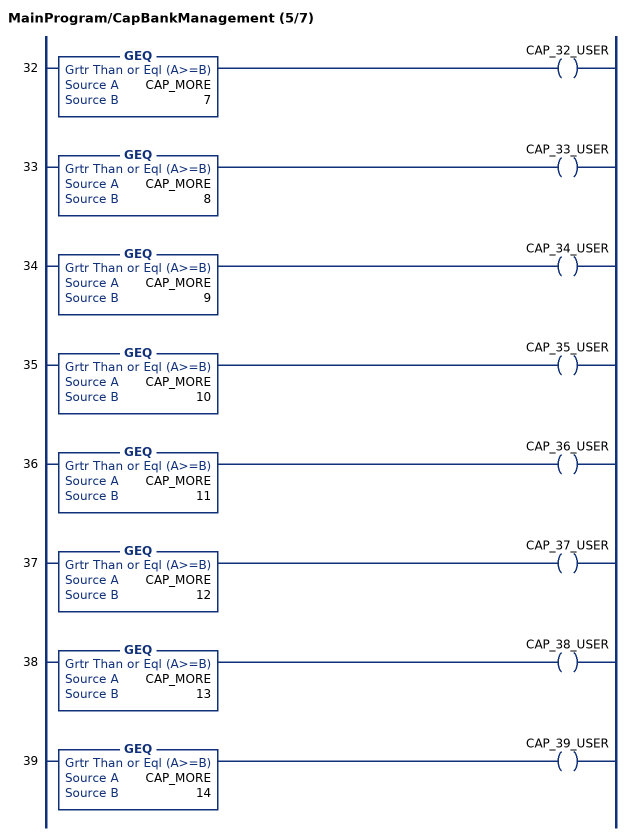
   32: GEQ(CAP_MORE,7)OTE(CAP_32_USER);
   33: GEQ(CAP_MORE,8)OTE(CAP_33_USER);
   34: GEQ(CAP_MORE,9)OTE(CAP_34_USER);
   35: GEQ(CAP_MORE,10)OTE(CAP_35_USER);
   36: GEQ(CAP_MORE,11)OTE(CAP_36_USER);
   37: GEQ(CAP_MORE,12)OTE(CAP_37_USER);
   38: GEQ(CAP_MORE,13)OTE(CAP_38_USER);
   39: GEQ(CAP_MORE,14)OTE(CAP_39_USER);
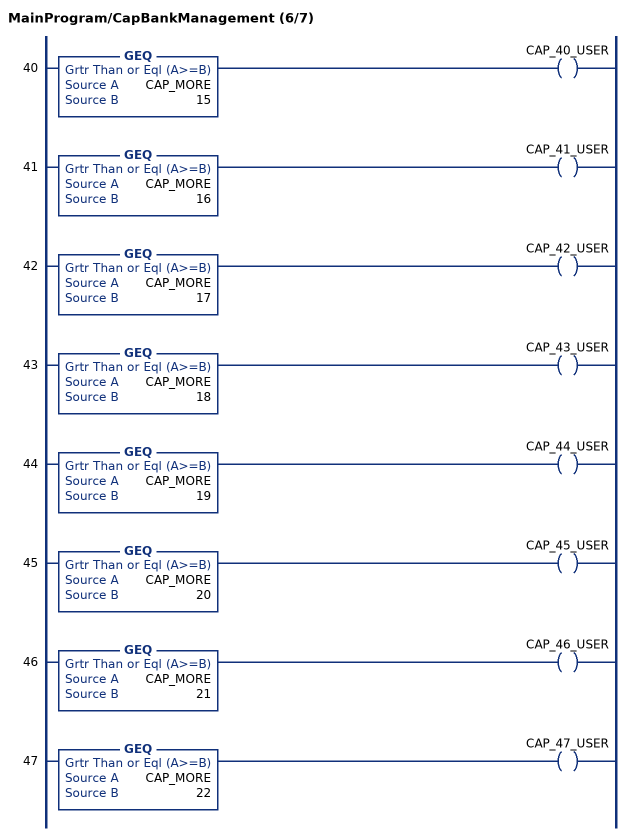
   40: GEQ(CAP_MORE,15)OTE(CAP_40_USER);
   41: GEQ(CAP_MORE,16)OTE(CAP_41_USER);
   42: GEQ(CAP_MORE,17)OTE(CAP_42_USER);
   43: GEQ(CAP_MORE,18)OTE(CAP_43_USER);
   44: GEQ(CAP_MORE,19)OTE(CAP_44_USER);
   45: GEQ(CAP_MORE,20)OTE(CAP_45_USER);
   46: GEQ(CAP_MORE,21)OTE(CAP_46_USER);
   47: GEQ(CAP_MORE,22)OTE(CAP_47_USER);
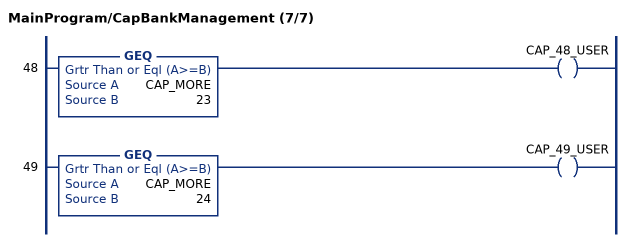
   48: GEQ(CAP_MORE,23)OTE(CAP_48_USER);
   49: GEQ(CAP_MORE,24)OTE(CAP_49_USER);
END_ROUTINE

ROUTINE CapBankOperation   (* ladder *)
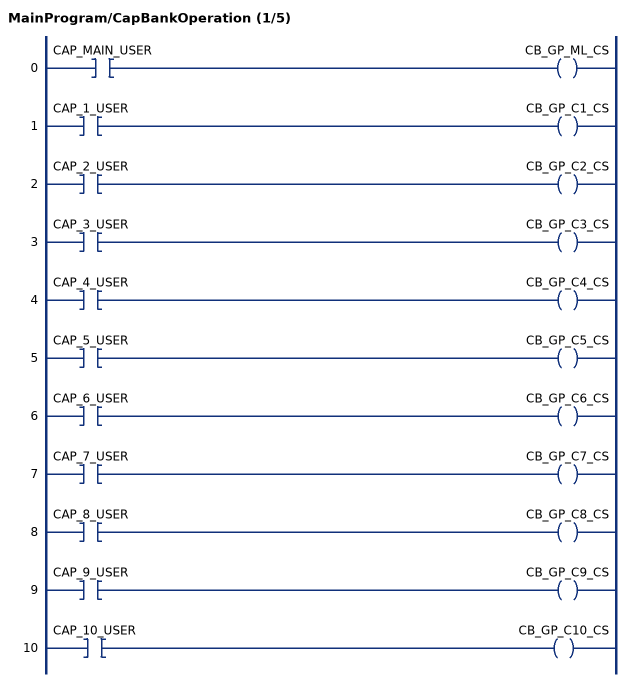
   0: XIC(CAP_MAIN_USER)OTE(CB_GP_ML_CS);
   1: XIC(CAP_1_USER)OTE(CB_GP_C1_CS);
   2: XIC(CAP_2_USER)OTE(CB_GP_C2_CS);
   3: XIC(CAP_3_USER)OTE(CB_GP_C3_CS);
   4: XIC(CAP_4_USER)OTE(CB_GP_C4_CS);
   5: XIC(CAP_5_USER)OTE(CB_GP_C5_CS);
   6: XIC(CAP_6_USER)OTE(CB_GP_C6_CS);
   7: XIC(CAP_7_USER)OTE(CB_GP_C7_CS);
   8: XIC(CAP_8_USER)OTE(CB_GP_C8_CS);
   9: XIC(CAP_9_USER)OTE(CB_GP_C9_CS);
   10: XIC(CAP_10_USER)OTE(CB_GP_C10_CS);
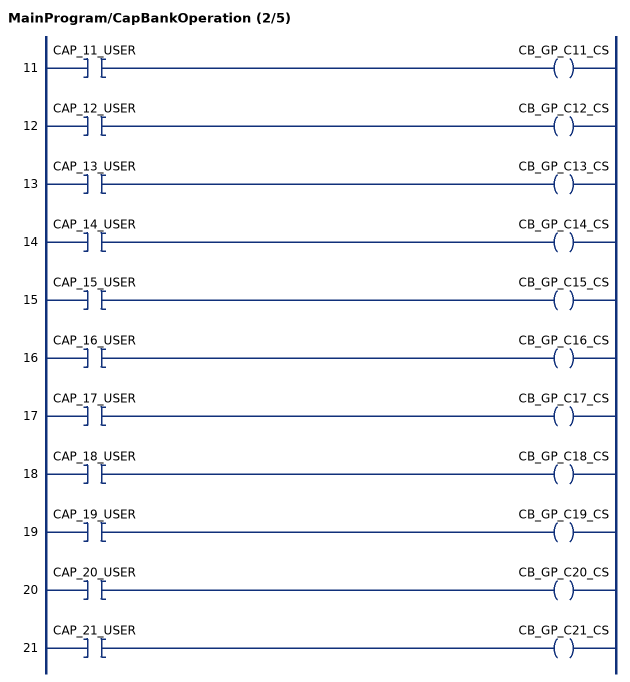
   11: XIC(CAP_11_USER)OTE(CB_GP_C11_CS);
   12: XIC(CAP_12_USER)OTE(CB_GP_C12_CS);
   13: XIC(CAP_13_USER)OTE(CB_GP_C13_CS);
   14: XIC(CAP_14_USER)OTE(CB_GP_C14_CS);
   15: XIC(CAP_15_USER)OTE(CB_GP_C15_CS);
   16: XIC(CAP_16_USER)OTE(CB_GP_C16_CS);
   17: XIC(CAP_17_USER)OTE(CB_GP_C17_CS);
   18: XIC(CAP_18_USER)OTE(CB_GP_C18_CS);
   19: XIC(CAP_19_USER)OTE(CB_GP_C19_CS);
   20: XIC(CAP_20_USER)OTE(CB_GP_C20_CS);
   21: XIC(CAP_21_USER)OTE(CB_GP_C21_CS);
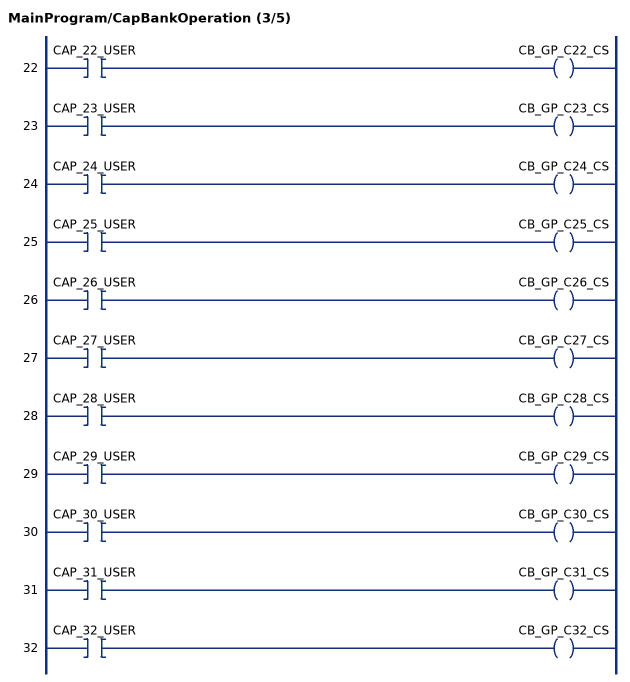
   22: XIC(CAP_22_USER)OTE(CB_GP_C22_CS);
   23: XIC(CAP_23_USER)OTE(CB_GP_C23_CS);
   24: XIC(CAP_24_USER)OTE(CB_GP_C24_CS);
   25: XIC(CAP_25_USER)OTE(CB_GP_C25_CS);
   26: XIC(CAP_26_USER)OTE(CB_GP_C26_CS);
   27: XIC(CAP_27_USER)OTE(CB_GP_C27_CS);
   28: XIC(CAP_28_USER)OTE(CB_GP_C28_CS);
   29: XIC(CAP_29_USER)OTE(CB_GP_C29_CS);
   30: XIC(CAP_30_USER)OTE(CB_GP_C30_CS);
   31: XIC(CAP_31_USER)OTE(CB_GP_C31_CS);
   32: XIC(CAP_32_USER)OTE(CB_GP_C32_CS);
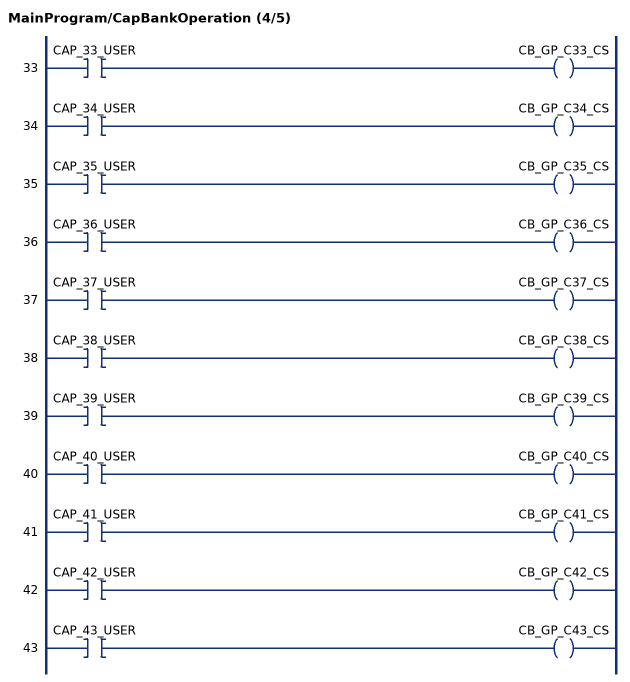
   33: XIC(CAP_33_USER)OTE(CB_GP_C33_CS);
   34: XIC(CAP_34_USER)OTE(CB_GP_C34_CS);
   35: XIC(CAP_35_USER)OTE(CB_GP_C35_CS);
   36: XIC(CAP_36_USER)OTE(CB_GP_C36_CS);
   37: XIC(CAP_37_USER)OTE(CB_GP_C37_CS);
   38: XIC(CAP_38_USER)OTE(CB_GP_C38_CS);
   39: XIC(CAP_39_USER)OTE(CB_GP_C39_CS);
   40: XIC(CAP_40_USER)OTE(CB_GP_C40_CS);
   41: XIC(CAP_41_USER)OTE(CB_GP_C41_CS);
   42: XIC(CAP_42_USER)OTE(CB_GP_C42_CS);
   43: XIC(CAP_43_USER)OTE(CB_GP_C43_CS);
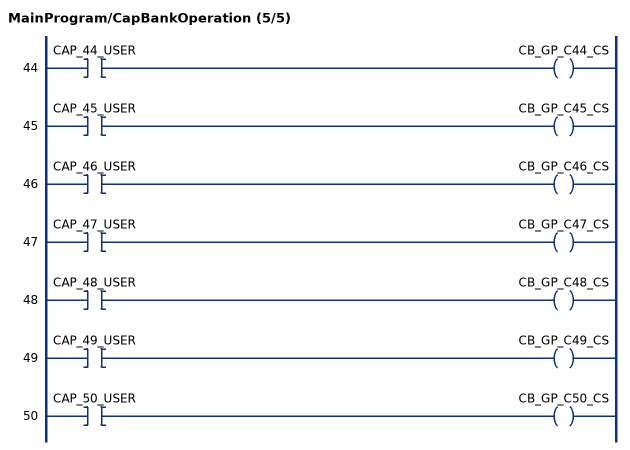
   44: XIC(CAP_44_USER)OTE(CB_GP_C44_CS);
   45: XIC(CAP_45_USER)OTE(CB_GP_C45_CS);
   46: XIC(CAP_46_USER)OTE(CB_GP_C46_CS);
   47: XIC(CAP_47_USER)OTE(CB_GP_C47_CS);
   48: XIC(CAP_48_USER)OTE(CB_GP_C48_CS);
   49: XIC(CAP_49_USER)OTE(CB_GP_C49_CS);
   50: XIC(CAP_50_USER)OTE(CB_GP_C50_CS);
END_ROUTINE

ROUTINE GridManagement   (* ladder *)
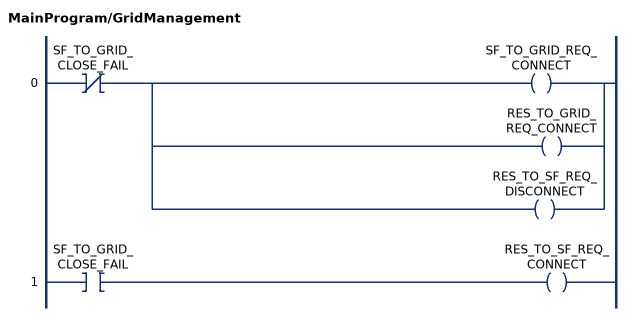
   0: XIO(SF_TO_GRID_CLOSE_FAIL)[OTE(SF_TO_GRID_REQ_CONNECT) ,OTE(RES_TO_GRID_REQ_CONNECT) ,OTE(RES_TO_SF_REQ_DISCONNECT) ];
   1: XIC(SF_TO_GRID_CLOSE_FAIL)OTE(RES_TO_SF_REQ_CONNECT);
END_ROUTINE

ROUTINE GridOperation   (* ladder *)
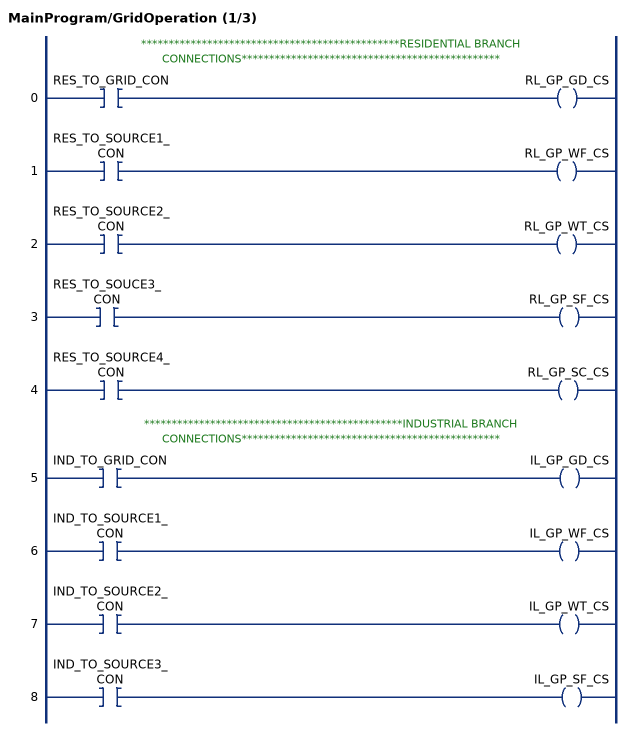
   // ***********************************************RESIDENTIAL BRANCH CONNECTIONS***********************************************
   0: XIC(RES_TO_GRID_CON)OTE(RL_GP_GD_CS);
   1: XIC(RES_TO_SOURCE1_CON)OTE(RL_GP_WF_CS);
   2: XIC(RES_TO_SOURCE2_CON)OTE(RL_GP_WT_CS);
   3: XIC(RES_TO_SOUCE3_CON)OTE(RL_GP_SF_CS);
   4: XIC(RES_TO_SOURCE4_CON)OTE(RL_GP_SC_CS);
   // ***********************************************INDUSTRIAL BRANCH CONNECTIONS***********************************************
   5: XIC(IND_TO_GRID_CON)OTE(IL_GP_GD_CS);
   6: XIC(IND_TO_SOURCE1_CON)OTE(IL_GP_WF_CS);
   7: XIC(IND_TO_SOURCE2_CON)OTE(IL_GP_WT_CS);
   8: XIC(IND_TO_SOURCE3_CON)OTE(IL_GP_SF_CS);
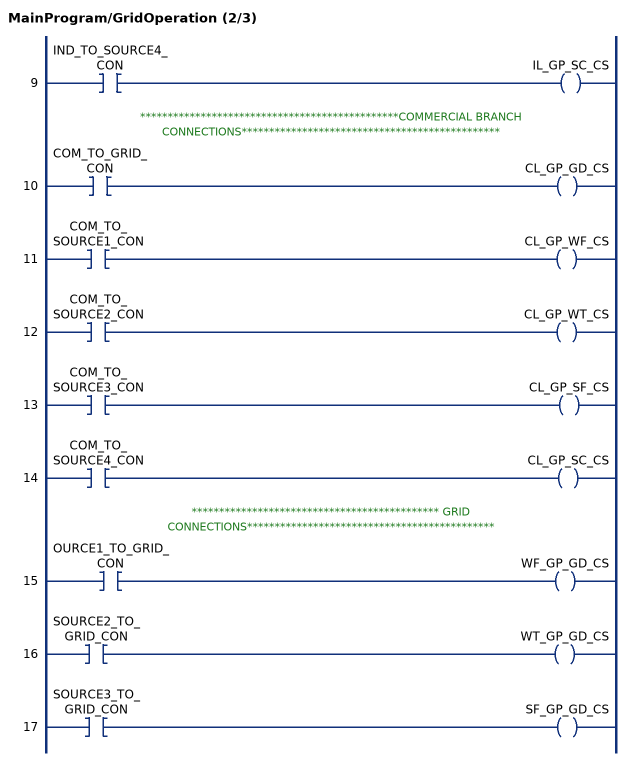
   9: XIC(IND_TO_SOURCE4_CON)OTE(IL_GP_SC_CS);
   // ***********************************************COMMERCIAL BRANCH CONNECTIONS***********************************************
   10: XIC(COM_TO_GRID_CON)OTE(CL_GP_GD_CS);
   11: XIC(COM_TO_SOURCE1_CON)OTE(CL_GP_WF_CS);
   12: XIC(COM_TO_SOURCE2_CON)OTE(CL_GP_WT_CS);
   13: XIC(COM_TO_SOURCE3_CON)OTE(CL_GP_SF_CS);
   14: XIC(COM_TO_SOURCE4_CON)OTE(CL_GP_SC_CS);
   // ********************************************* GRID CONNECTIONS*********************************************
   15: XIC(OURCE1_TO_GRID_CON)OTE(WF_GP_GD_CS);
   16: XIC(SOURCE2_TO_GRID_CON)OTE(WT_GP_GD_CS);
   17: XIC(SOURCE3_TO_GRID_CON)OTE(SF_GP_GD_CS);
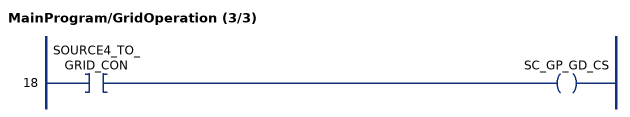
   18: XIC(SOURCE4_TO_GRID_CON)OTE(SC_GP_GD_CS);
END_ROUTINE

ROUTINE IMPORT_DATA   (* ladder *)
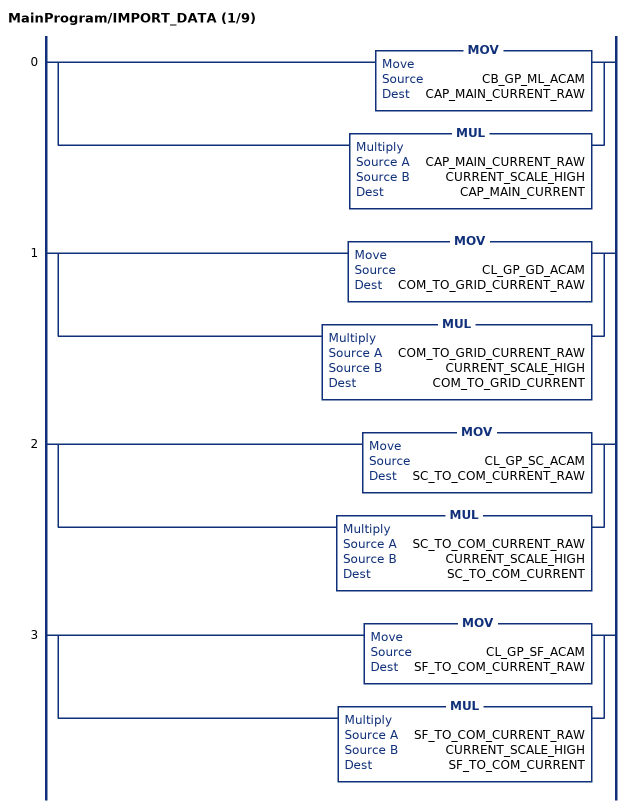
   0: [MOV(CB_GP_ML_ACAM,CAP_MAIN_CURRENT_RAW) ,MUL(CAP_MAIN_CURRENT_RAW,CURRENT_SCALE_HIGH,CAP_MAIN_CURRENT) ];
   1: [MOV(CL_GP_GD_ACAM,COM_TO_GRID_CURRENT_RAW) ,MUL(COM_TO_GRID_CURRENT_RAW,CURRENT_SCALE_HIGH,COM_TO_GRID_CURRENT) ];
   2: [MOV(CL_GP_SC_ACAM,SC_TO_COM_CURRENT_RAW) ,MUL(SC_TO_COM_CURRENT_RAW,CURRENT_SCALE_HIGH,SC_TO_COM_CURRENT) ];
   3: [MOV(CL_GP_SF_ACAM,SF_TO_COM_CURRENT_RAW) ,MUL(SF_TO_COM_CURRENT_RAW,CURRENT_SCALE_HIGH,SF_TO_COM_CURRENT) ];
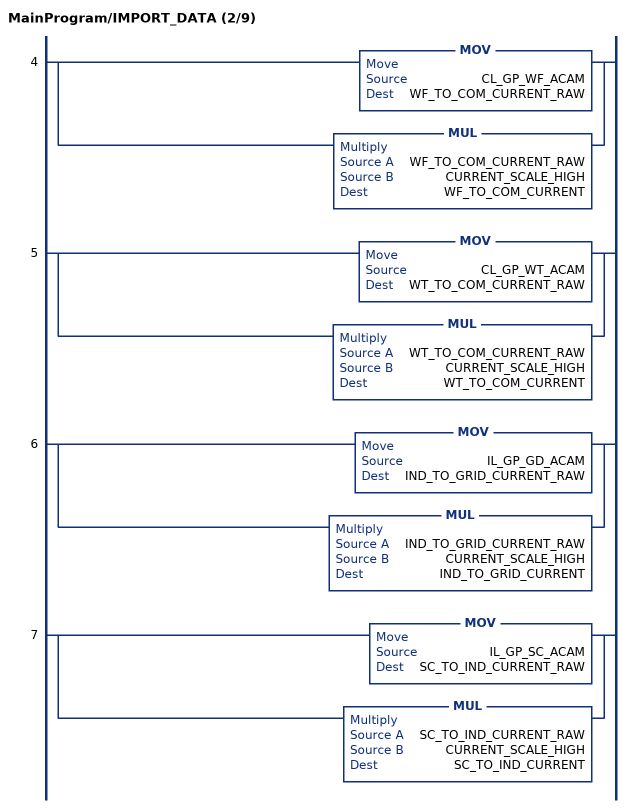
   4: [MOV(CL_GP_WF_ACAM,WF_TO_COM_CURRENT_RAW) ,MUL(WF_TO_COM_CURRENT_RAW,CURRENT_SCALE_HIGH,WF_TO_COM_CURRENT) ];
   5: [MOV(CL_GP_WT_ACAM,WT_TO_COM_CURRENT_RAW) ,MUL(WT_TO_COM_CURRENT_RAW,CURRENT_SCALE_HIGH,WT_TO_COM_CURRENT) ];
   6: [MOV(IL_GP_GD_ACAM,IND_TO_GRID_CURRENT_RAW) ,MUL(IND_TO_GRID_CURRENT_RAW,CURRENT_SCALE_HIGH,IND_TO_GRID_CURRENT) ];
   7: [MOV(IL_GP_SC_ACAM,SC_TO_IND_CURRENT_RAW) ,MUL(SC_TO_IND_CURRENT_RAW,CURRENT_SCALE_HIGH,SC_TO_IND_CURRENT) ];
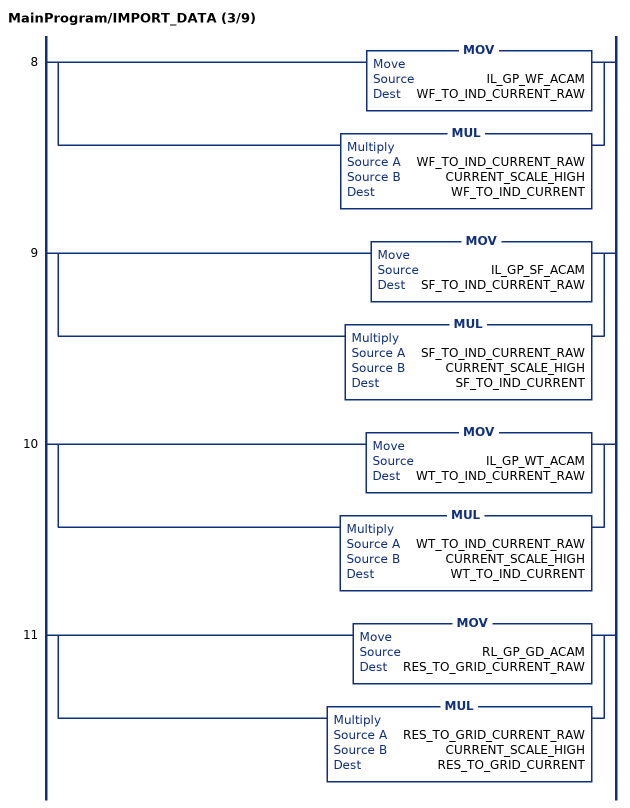
   8: [MOV(IL_GP_WF_ACAM,WF_TO_IND_CURRENT_RAW) ,MUL(WF_TO_IND_CURRENT_RAW,CURRENT_SCALE_HIGH,WF_TO_IND_CURRENT) ];
   9: [MOV(IL_GP_SF_ACAM,SF_TO_IND_CURRENT_RAW) ,MUL(SF_TO_IND_CURRENT_RAW,CURRENT_SCALE_HIGH,SF_TO_IND_CURRENT) ];
   10: [MOV(IL_GP_WT_ACAM,WT_TO_IND_CURRENT_RAW) ,MUL(WT_TO_IND_CURRENT_RAW,CURRENT_SCALE_HIGH,WT_TO_IND_CURRENT) ];
   11: [MOV(RL_GP_GD_ACAM,RES_TO_GRID_CURRENT_RAW) ,MUL(RES_TO_GRID_CURRENT_RAW,CURRENT_SCALE_HIGH,RES_TO_GRID_CURRENT) ];
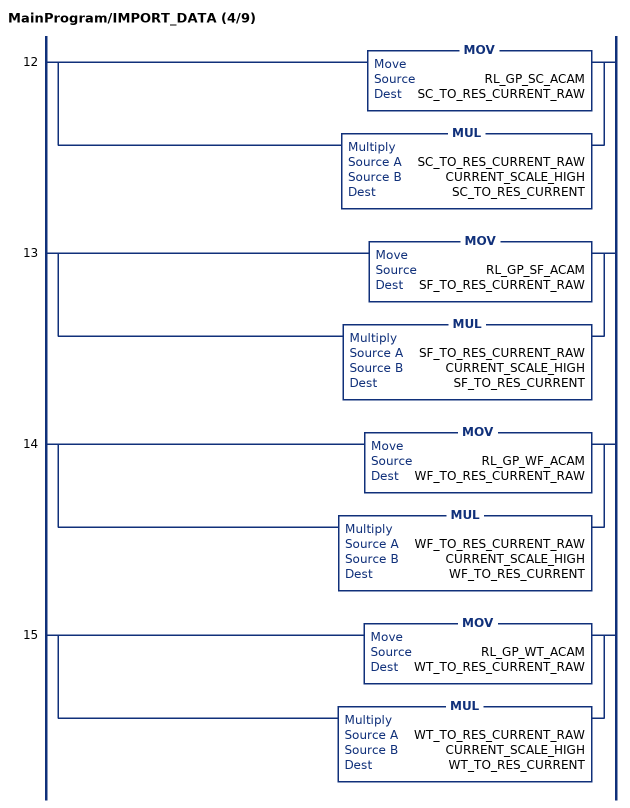
   12: [MOV(RL_GP_SC_ACAM,SC_TO_RES_CURRENT_RAW) ,MUL(SC_TO_RES_CURRENT_RAW,CURRENT_SCALE_HIGH,SC_TO_RES_CURRENT) ];
   13: [MOV(RL_GP_SF_ACAM,SF_TO_RES_CURRENT_RAW) ,MUL(SF_TO_RES_CURRENT_RAW,CURRENT_SCALE_HIGH,SF_TO_RES_CURRENT) ];
   14: [MOV(RL_GP_WF_ACAM,WF_TO_RES_CURRENT_RAW) ,MUL(WF_TO_RES_CURRENT_RAW,CURRENT_SCALE_HIGH,WF_TO_RES_CURRENT) ];
   15: [MOV(RL_GP_WT_ACAM,WT_TO_RES_CURRENT_RAW) ,MUL(WT_TO_RES_CURRENT_RAW,CURRENT_SCALE_HIGH,WT_TO_RES_CURRENT) ];
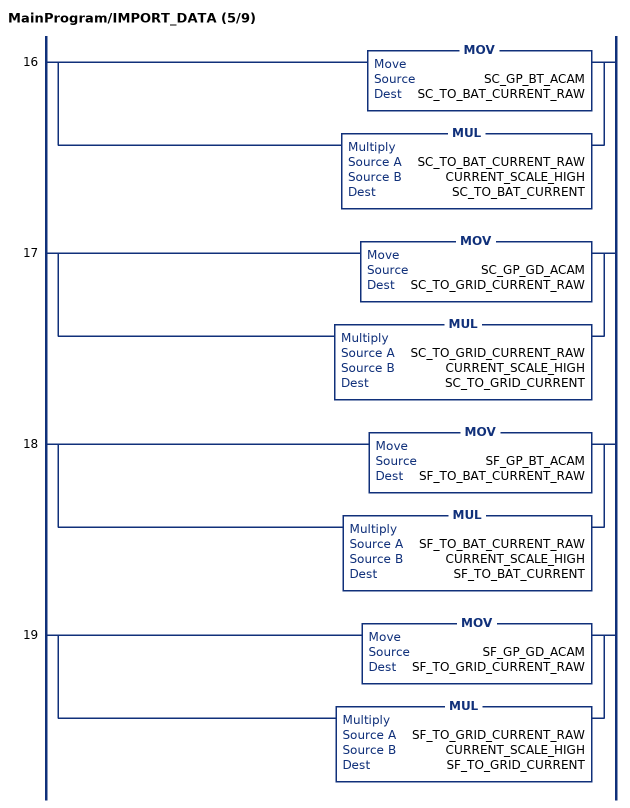
   16: [MOV(SC_GP_BT_ACAM,SC_TO_BAT_CURRENT_RAW) ,MUL(SC_TO_BAT_CURRENT_RAW,CURRENT_SCALE_HIGH,SC_TO_BAT_CURRENT) ];
   17: [MOV(SC_GP_GD_ACAM,SC_TO_GRID_CURRENT_RAW) ,MUL(SC_TO_GRID_CURRENT_RAW,CURRENT_SCALE_HIGH,SC_TO_GRID_CURRENT) ];
   18: [MOV(SF_GP_BT_ACAM,SF_TO_BAT_CURRENT_RAW) ,MUL(SF_TO_BAT_CURRENT_RAW,CURRENT_SCALE_HIGH,SF_TO_BAT_CURRENT) ];
   19: [MOV(SF_GP_GD_ACAM,SF_TO_GRID_CURRENT_RAW) ,MUL(SF_TO_GRID_CURRENT_RAW,CURRENT_SCALE_HIGH,SF_TO_GRID_CURRENT) ];
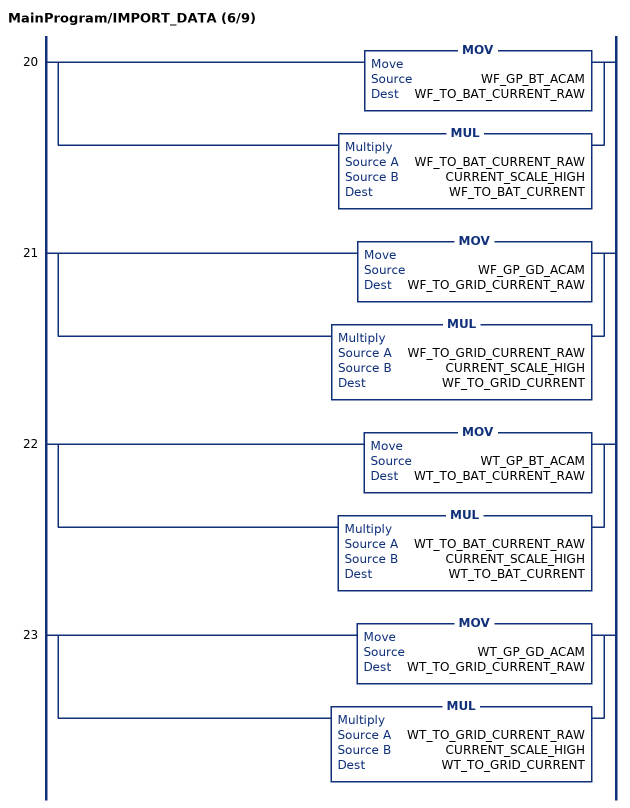
   20: [MOV(WF_GP_BT_ACAM,WF_TO_BAT_CURRENT_RAW) ,MUL(WF_TO_BAT_CURRENT_RAW,CURRENT_SCALE_HIGH,WF_TO_BAT_CURRENT) ];
   21: [MOV(WF_GP_GD_ACAM,WF_TO_GRID_CURRENT_RAW) ,MUL(WF_TO_GRID_CURRENT_RAW,CURRENT_SCALE_HIGH,WF_TO_GRID_CURRENT) ];
   22: [MOV(WT_GP_BT_ACAM,WT_TO_BAT_CURRENT_RAW) ,MUL(WT_TO_BAT_CURRENT_RAW,CURRENT_SCALE_HIGH,WT_TO_BAT_CURRENT) ];
   23: [MOV(WT_GP_GD_ACAM,WT_TO_GRID_CURRENT_RAW) ,MUL(WT_TO_GRID_CURRENT_RAW,CURRENT_SCALE_HIGH,WT_TO_GRID_CURRENT) ];
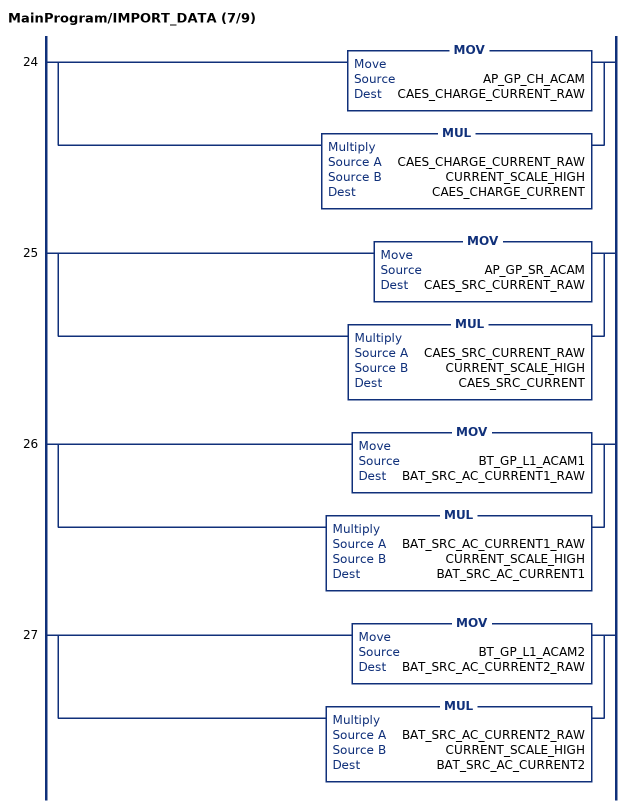
   24: [MOV(AP_GP_CH_ACAM,CAES_CHARGE_CURRENT_RAW) ,MUL(CAES_CHARGE_CURRENT_RAW,CURRENT_SCALE_HIGH,CAES_CHARGE_CURRENT) ];
   25: [MOV(AP_GP_SR_ACAM,CAES_SRC_CURRENT_RAW) ,MUL(CAES_SRC_CURRENT_RAW,CURRENT_SCALE_HIGH,CAES_SRC_CURRENT) ];
   26: [MOV(BT_GP_L1_ACAM1,BAT_SRC_AC_CURRENT1_RAW) ,MUL(BAT_SRC_AC_CURRENT1_RAW,CURRENT_SCALE_HIGH,BAT_SRC_AC_CURRENT1) ];
   27: [MOV(BT_GP_L1_ACAM2,BAT_SRC_AC_CURRENT2_RAW) ,MUL(BAT_SRC_AC_CURRENT2_RAW,CURRENT_SCALE_HIGH,BAT_SRC_AC_CURRENT2) ];
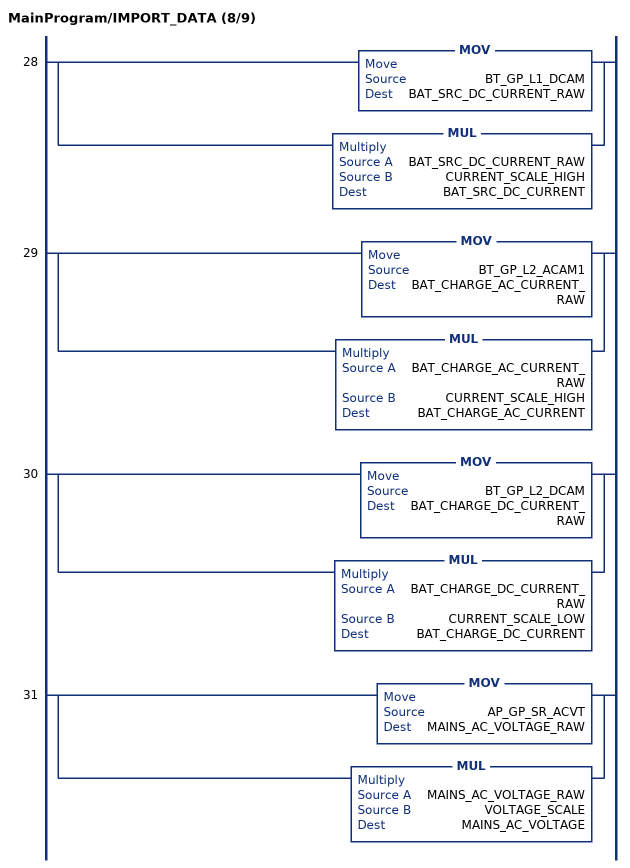
   28: [MOV(BT_GP_L1_DCAM,BAT_SRC_DC_CURRENT_RAW) ,MUL(BAT_SRC_DC_CURRENT_RAW,CURRENT_SCALE_HIGH,BAT_SRC_DC_CURRENT) ];
   29: [MOV(BT_GP_L2_ACAM1,BAT_CHARGE_AC_CURRENT_RAW) ,MUL(BAT_CHARGE_AC_CURRENT_RAW,CURRENT_SCALE_HIGH,BAT_CHARGE_AC_CURRENT) ];
   30: [MOV(BT_GP_L2_DCAM,BAT_CHARGE_DC_CURRENT_RAW) ,MUL(BAT_CHARGE_DC_CURRENT_RAW,CURRENT_SCALE_LOW,BAT_CHARGE_DC_CURRENT) ];
   31: [MOV(AP_GP_SR_ACVT,MAINS_AC_VOLTAGE_RAW) ,MUL(MAINS_AC_VOLTAGE_RAW,VOLTAGE_SCALE,MAINS_AC_VOLTAGE) ];
